   PLI_EC[144] := FALSE;
   PLI_EC[145] := FALSE;
   PLI_EC[146] := FALSE;
   PLI_EC[147] := FALSE;
   PLI_EC[148] := FALSE;
   PLI_EC[149] := FALSE;
   PLI_EC[150] := FALSE;
   PLI_R[1] := FALSE;
   PLI_R[2] := FALSE;
   PLI_R[3] := FALSE;
   PLI_R[4] := FALSE;
   PLI_R[5] := FALSE;
   PLI_R[6] := FALSE;
   PLI_R[7] := FALSE;
   PLI_R[8] := FALSE;
   PLI_R[9] := FALSE;
   PLI_R[10] := FALSE;
   PLI_R[11] := FALSE;
   PLI_R[12] := FALSE;
   PLI_R[13] := FALSE;
   PLI_R[14] := FALSE;
   PLI_R[15] := FALSE;
   PLI_R[16] := FALSE;
   PLI_R[17] := FALSE;
   PLI_R[18] := FALSE;
   PLI_R[19] := FALSE;
   PLI_R[20] := FALSE;
   PLI_R[21] := FALSE;
   PLI_R[22] := FALSE;
   PLI_R[23] := FALSE;
   PLI_R[24] := FALSE;
   PLI_R[25] := FALSE;
   PLI_R[26] := FALSE;
   PLI_R[27] := FALSE;
   PLI_R[28] := FALSE;
   PLI_R[29] := FALSE;
   PLI_R[30] := FALSE;
   PLI_R[31] := FALSE;
   PLI_R[32] := FALSE;
   PLI_R[33] := FALSE;
   PLI_R[34] := FALSE;
   PLI_R[35] := FALSE;
   PLI_R[36] := FALSE;
   PLI_R[37] := FALSE;
   PLI_R[38] := FALSE;
   PLI_R[39] := FALSE;
   PLI_R[40] := FALSE;
   PLI_R[41] := FALSE;
   PLI_R[42] := FALSE;
   PLI_R[43] := FALSE;
   PLI_R[44] := TRUE;
   PLI_R[45] := FALSE;
   PLI_R[46] := FALSE;
   PLI_R[47] := FALSE;
   PLI_R[48] := FALSE;
   PLI_R[49] := FALSE;
   PLI_R[50] := FALSE;
   PLI_R[51] := FALSE;
   PLI_R[52] := FALSE;
   PLI_R[53] := FALSE;
   PLI_R[54] := FALSE;
   PLI_R[55] := FALSE;
   PLI_R[56] := FALSE;
   PLI_R[57] := FALSE;
   PLI_R[58] := FALSE;
   PLI_R[59] := FALSE;
   PLI_R[60] := FALSE;
   PLI_R[61] := FALSE;
   PLI_R[62] := FALSE;
   PLI_R[63] := FALSE;
   PLI_R[64] := FALSE;
   PLI_R[65] := FALSE;
   PLI_R[66] := FALSE;
   PLI_R[67] := FALSE;
   PLI_R[68] := FALSE;
   PLI_R[69] := FALSE;
   PLI_R[70] := FALSE;
   PLI_R[71] := FALSE;
   PLI_R[72] := FALSE;
   PLI_R[73] := FALSE;
   PLI_R[74] := FALSE;
   PLI_R[75] := FALSE;
   PLI_R[76] := FALSE;
   PLI_R[77] := FALSE;
   PLI_R[78] := FALSE;
   PLI_R[79] := FALSE;
   PLI_R[80] := FALSE;
   PLI_R[81] := FALSE;
   PLI_R[82] := FALSE;
   PLI_R[83] := FALSE;
   PLI_R[84] := FALSE;
   PLI_R[85] := FALSE;
   PLI_R[86] := FALSE;
   PLI_R[87] := FALSE;
   PLI_R[88] := FALSE;
   PLI_R[89] := FALSE;
   PLI_R[90] := FALSE;
   PLI_R[91] := FALSE;
   PLI_R[92] := FALSE;
   PLI_R[93] := FALSE;
   PLI_R[94] := FALSE;
   PLI_R[95] := FALSE;
   PLI_R[96] := FALSE;
   PLI_R[97] := FALSE;
   PLI_R[98] := FALSE;
   PLI_R[99] := FALSE;
   PLI_R[100] := FALSE;
   PLI_R[101] := FALSE;
   PLI_R[102] := FALSE;
   PLI_R[103] := FALSE;
   PLI_R[104] := FALSE;
   PLI_R[105] := FALSE;
   PLI_R[106] := FALSE;
   PLI_R[107] := FALSE;
   PLI_R[108] := FALSE;
   PLI_R[109] := FALSE;
   PLI_R[110] := TRUE;
   PLI_R[111] := TRUE;
   PLI_R[112] := FALSE;
   PLI_R[113] := FALSE;
   PLI_R[114] := FALSE;
   PLI_R[115] := FALSE;
   PLI_R[116] := TRUE;
   PLI_R[117] := FALSE;
   PLI_R[118] := FALSE;
   PLI_R[119] := FALSE;
   PLI_R[120] := FALSE;
   PLI_R[121] := FALSE;
   PLI_R[122] := FALSE;
   PLI_R[123] := FALSE;
   PLI_R[124] := FALSE;
   PLI_R[125] := FALSE;
   PLI_R[126] := FALSE;
   PLI_R[127] := FALSE;
   PLI_R[128] := FALSE;
   PLI_R[129] := FALSE;
   PLI_R[130] := FALSE;
   PLI_R[131] := FALSE;
   PLI_R[132] := FALSE;
   PLI_R[133] := FALSE;
   PLI_R[134] := FALSE;
   PLI_R[135] := FALSE;
   PLI_R[136] := FALSE;
   PLI_R[137] := FALSE;
   PLI_R[138] := FALSE;
   PLI_R[139] := FALSE;
   PLI_R[140] := FALSE;
   PLI_R[141] := FALSE;
   PLI_R[142] := FALSE;
   PLI_R[143] := FALSE;
   PLI_R[144] := FALSE;
   PLI_R[145] := FALSE;
   PLI_R[146] := FALSE;
   PLI_R[147] := FALSE;
   PLI_R[148] := FALSE;
   PLI_R[149] := FALSE;
   PLI_R[150] := FALSE;
   PLI_T[1] := FALSE;
   PLI_T[2] := FALSE;
   PLI_T[3] := FALSE;
   PLI_T[4] := FALSE;
   PLI_T[5] := FALSE;
   PLI_T[6] := FALSE;
   PLI_T[7] := FALSE;
   PLI_T[8] := FALSE;
   PLI_T[9] := FALSE;
   PLI_T[10] := FALSE;
   PLI_T[11] := FALSE;
   PLI_T[12] := FALSE;
   PLI_T[13] := FALSE;
   PLI_T[14] := FALSE;
   PLI_T[15] := FALSE;
   PLI_T[16] := FALSE;
   PLI_T[17] := FALSE;
   PLI_T[18] := FALSE;
   PLI_T[19] := FALSE;
   PLI_T[20] := FALSE;
   PLI_T[21] := FALSE;
   PLI_T[22] := FALSE;
   PLI_T[23] := FALSE;
   PLI_T[24] := FALSE;
   PLI_T[25] := FALSE;
   PLI_T[26] := FALSE;
   PLI_T[27] := FALSE;
   PLI_T[28] := FALSE;
   PLI_T[29] := FALSE;
   PLI_T[30] := FALSE;
   PLI_T[31] := FALSE;
   PLI_T[32] := FALSE;
   PLI_T[33] := FALSE;
   PLI_T[34] := FALSE;
   PLI_T[35] := FALSE;
   PLI_T[36] := FALSE;
   PLI_T[37] := FALSE;
   PLI_T[38] := FALSE;
   PLI_T[39] := FALSE;
   PLI_T[40] := FALSE;
   PLI_T[41] := FALSE;
   PLI_T[42] := FALSE;
   PLI_T[43] := FALSE;
   PLI_T[44] := FALSE;
   PLI_T[45] := FALSE;
   PLI_T[46] := FALSE;
   PLI_T[47] := FALSE;
   PLI_T[48] := FALSE;
   PLI_T[49] := FALSE;
   PLI_T[50] := FALSE;
   PLI_T[51] := FALSE;
   PLI_T[52] := FALSE;
   PLI_T[53] := FALSE;
   PLI_T[54] := FALSE;
   PLI_T[55] := FALSE;
   PLI_T[56] := FALSE;
   PLI_T[57] := FALSE;
   PLI_T[58] := FALSE;
   PLI_T[59] := FALSE;
   PLI_T[60] := FALSE;
   PLI_T[61] := FALSE;
   PLI_T[62] := FALSE;
   PLI_T[63] := FALSE;
   PLI_T[64] := FALSE;
   PLI_T[65] := FALSE;
   PLI_T[66] := FALSE;
   PLI_T[67] := FALSE;
   PLI_T[68] := FALSE;
   PLI_T[69] := FALSE;
   PLI_T[70] := FALSE;
   PLI_T[71] := FALSE;
   PLI_T[72] := FALSE;
   PLI_T[73] := FALSE;
   PLI_T[74] := FALSE;
   PLI_T[75] := FALSE;
   PLI_T[76] := FALSE;
   PLI_T[77] := FALSE;
   PLI_T[78] := FALSE;
   PLI_T[79] := FALSE;
   PLI_T[80] := FALSE;
   PLI_T[81] := FALSE;
   PLI_T[82] := FALSE;
   PLI_T[83] := FALSE;
   PLI_T[84] := FALSE;
   PLI_T[85] := FALSE;
   PLI_T[86] := FALSE;
   PLI_T[87] := FALSE;
   PLI_T[88] := FALSE;
   PLI_T[89] := FALSE;
   PLI_T[90] := FALSE;
   PLI_T[91] := FALSE;
   PLI_T[92] := FALSE;
   PLI_T[93] := FALSE;
   PLI_T[94] := FALSE;
   PLI_T[95] := FALSE;
   PLI_T[96] := FALSE;
   PLI_T[97] := FALSE;
   PLI_T[98] := FALSE;
   PLI_T[99] := FALSE;
   PLI_T[100] := FALSE;
   PLI_T[101] := FALSE;
   PLI_T[102] := FALSE;
   PLI_T[103] := FALSE;
   PLI_T[104] := FALSE;
   PLI_T[105] := FALSE;
   PLI_T[106] := FALSE;
   PLI_T[107] := FALSE;
   PLI_T[108] := FALSE;
   PLI_T[109] := FALSE;
   PLI_T[110] := FALSE;
   PLI_T[111] := FALSE;
   PLI_T[112] := FALSE;
   PLI_T[113] := FALSE;
   PLI_T[114] := FALSE;
   PLI_T[115] := FALSE;
   PLI_T[116] := FALSE;
   PLI_T[117] := FALSE;
   PLI_T[118] := FALSE;
   PLI_T[119] := FALSE;
   PLI_T[120] := FALSE;
   PLI_T[121] := FALSE;
   PLI_T[122] := FALSE;
   PLI_T[123] := FALSE;
   PLI_T[124] := FALSE;
   PLI_T[125] := FALSE;
   PLI_T[126] := FALSE;
   PLI_T[127] := FALSE;
   PLI_T[128] := FALSE;
   PLI_T[129] := FALSE;
   PLI_T[130] := FALSE;
   PLI_T[131] := FALSE;
   PLI_T[132] := FALSE;
   PLI_T[133] := FALSE;
   PLI_T[134] := FALSE;
   PLI_T[135] := FALSE;
   PLI_T[136] := FALSE;
   PLI_T[137] := FALSE;
   PLI_T[138] := FALSE;
   PLI_T[139] := FALSE;
   PLI_T[140] := FALSE;
   PLI_T[141] := FALSE;
   PLI_T[142] := FALSE;
   PLI_T[143] := FALSE;
   PLI_T[144] := FALSE;
   PLI_T[145] := FALSE;
   PLI_T[146] := FALSE;
   PLI_T[147] := FALSE;
   PLI_T[148] := FALSE;
   PLI_T[149] := FALSE;
   PLI_T[150] := FALSE;
   PLI_A[1] := FALSE;
   PLI_A[2] := FALSE;
   PLI_A[3] := FALSE;
   PLI_A[4] := FALSE;
   PLI_A[5] := FALSE;
   PLI_A[6] := FALSE;
   PLI_A[7] := FALSE;
   PLI_A[8] := FALSE;
   PLI_A[9] := FALSE;
   PLI_A[10] := FALSE;
   PLI_A[11] := FALSE;
   PLI_A[12] := FALSE;
   PLI_A[13] := FALSE;
   PLI_A[14] := FALSE;
   PLI_A[15] := FALSE;
   PLI_A[16] := FALSE;
   PLI_A[17] := FALSE;
   PLI_A[18] := FALSE;
   PLI_A[19] := FALSE;
   PLI_A[20] := FALSE;
   PLI_A[21] := FALSE;
   PLI_A[22] := FALSE;
   PLI_A[23] := FALSE;
   PLI_A[24] := FALSE;
   PLI_A[25] := FALSE;
   PLI_A[26] := FALSE;
   PLI_A[27] := FALSE;
   PLI_A[28] := FALSE;
   PLI_A[29] := FALSE;
   PLI_A[30] := FALSE;
   PLI_A[31] := FALSE;
   PLI_A[32] := FALSE;
   PLI_A[33] := FALSE;
   PLI_A[34] := FALSE;
   PLI_A[35] := FALSE;
   PLI_A[36] := FALSE;
   PLI_A[37] := FALSE;
   PLI_A[38] := FALSE;
   PLI_A[39] := FALSE;
   PLI_A[40] := FALSE;
   PLI_A[41] := FALSE;
   PLI_A[42] := FALSE;
   PLI_A[43] := FALSE;
   PLI_A[44] := FALSE;
   PLI_A[45] := FALSE;
   PLI_A[46] := FALSE;
   PLI_A[47] := FALSE;
   PLI_A[48] := FALSE;
   PLI_A[49] := FALSE;
   PLI_A[50] := FALSE;
   PLI_A[51] := FALSE;
   PLI_A[52] := FALSE;
   PLI_A[53] := FALSE;
   PLI_A[54] := FALSE;
   PLI_A[55] := FALSE;
   PLI_A[56] := FALSE;
   PLI_A[57] := FALSE;
   PLI_A[58] := FALSE;
   PLI_A[59] := FALSE;
   PLI_A[60] := FALSE;
   PLI_A[61] := FALSE;
   PLI_A[62] := FALSE;
   PLI_A[63] := FALSE;
   PLI_A[64] := FALSE;
   PLI_A[65] := FALSE;
   PLI_A[66] := FALSE;
   PLI_A[67] := FALSE;
   PLI_A[68] := FALSE;
   PLI_A[69] := FALSE;
   PLI_A[70] := FALSE;
   PLI_A[71] := FALSE;
   PLI_A[72] := FALSE;
   PLI_A[73] := FALSE;
   PLI_A[74] := FALSE;
   PLI_A[75] := FALSE;
   PLI_A[76] := FALSE;
   PLI_A[77] := FALSE;
   PLI_A[78] := FALSE;
   PLI_A[79] := FALSE;
   PLI_A[80] := FALSE;
   PLI_A[81] := FALSE;
   PLI_A[82] := FALSE;
   PLI_A[83] := FALSE;
   PLI_A[84] := FALSE;
   PLI_A[85] := FALSE;
   PLI_A[86] := FALSE;
   PLI_A[87] := FALSE;
   PLI_A[88] := FALSE;
   PLI_A[89] := FALSE;
   PLI_A[90] := FALSE;
   PLI_A[91] := FALSE;
   PLI_A[92] := FALSE;
   PLI_A[93] := FALSE;
   PLI_A[94] := FALSE;
   PLI_A[95] := FALSE;
   PLI_A[96] := FALSE;
   PLI_A[97] := FALSE;
   PLI_A[98] := FALSE;
   PLI_A[99] := FALSE;
   PLI_A[100] := FALSE;
   PLI_A[101] := FALSE;
   PLI_A[102] := FALSE;
   PLI_A[103] := FALSE;
   PLI_A[104] := FALSE;
   PLI_A[105] := FALSE;
   PLI_A[106] := FALSE;
   PLI_A[107] := FALSE;
   PLI_A[108] := FALSE;
   PLI_A[109] := FALSE;
   PLI_A[110] := FALSE;
   PLI_A[111] := FALSE;
   PLI_A[112] := FALSE;
   PLI_A[113] := FALSE;
   PLI_A[114] := FALSE;
   PLI_A[115] := FALSE;
   PLI_A[116] := FALSE;
   PLI_A[117] := FALSE;
   PLI_A[118] := FALSE;
   PLI_A[119] := FALSE;
   PLI_A[120] := FALSE;
   PLI_A[121] := FALSE;
   PLI_A[122] := FALSE;
   PLI_A[123] := FALSE;
   PLI_A[124] := FALSE;
   PLI_A[125] := FALSE;
   PLI_A[126] := FALSE;
   PLI_A[127] := FALSE;
   PLI_A[128] := FALSE;
   PLI_A[129] := FALSE;
   PLI_A[130] := FALSE;
   PLI_A[131] := FALSE;
   PLI_A[132] := FALSE;
   PLI_A[133] := FALSE;
   PLI_A[134] := FALSE;
   PLI_A[135] := FALSE;
   PLI_A[136] := FALSE;
   PLI_A[137] := FALSE;
   PLI_A[138] := FALSE;
   PLI_A[139] := FALSE;
   PLI_A[140] := FALSE;
   PLI_A[141] := FALSE;
   PLI_A[142] := FALSE;
   PLI_A[143] := FALSE;
   PLI_A[144] := FALSE;
   PLI_A[145] := FALSE;
   PLI_A[146] := FALSE;
   PLI_A[147] := FALSE;
   PLI_A[148] := FALSE;
   PLI_A[149] := FALSE;
   PLI_A[150] := FALSE;
   PLI_H[1] := FALSE;
   PLI_H[2] := FALSE;
   PLI_H[3] := FALSE;
   PLI_H[4] := FALSE;
   PLI_H[5] := FALSE;
   PLI_H[6] := FALSE;
   PLI_H[7] := FALSE;
   PLI_H[8] := FALSE;
   PLI_H[9] := FALSE;
   PLI_H[10] := FALSE;
   PLI_H[11] := FALSE;
   PLI_H[12] := FALSE;
   PLI_H[13] := FALSE;
   PLI_H[14] := FALSE;
   PLI_H[15] := FALSE;
   PLI_H[16] := FALSE;
   PLI_H[17] := FALSE;
   PLI_H[18] := FALSE;
   PLI_H[19] := FALSE;
   PLI_H[20] := FALSE;
   PLI_H[21] := FALSE;
   PLI_H[22] := FALSE;
   PLI_H[23] := FALSE;
   PLI_H[24] := FALSE;
   PLI_H[25] := FALSE;
   PLI_H[26] := FALSE;
   PLI_H[27] := FALSE;
   PLI_H[28] := FALSE;
   PLI_H[29] := FALSE;
   PLI_H[30] := FALSE;
   PLI_H[31] := FALSE;
   PLI_H[32] := FALSE;
   PLI_H[33] := FALSE;
   PLI_H[34] := FALSE;
   PLI_H[35] := FALSE;
   PLI_H[36] := FALSE;
   PLI_H[37] := FALSE;
   PLI_H[38] := FALSE;
   PLI_H[39] := FALSE;
   PLI_H[40] := FALSE;
   PLI_H[41] := FALSE;
   PLI_H[42] := FALSE;
   PLI_H[43] := FALSE;
   PLI_H[44] := FALSE;
   PLI_H[45] := FALSE;
   PLI_H[46] := FALSE;
   PLI_H[47] := FALSE;
   PLI_H[48] := FALSE;
   PLI_H[49] := FALSE;
   PLI_H[50] := FALSE;
   PLI_H[51] := FALSE;
   PLI_H[52] := FALSE;
   PLI_H[53] := FALSE;
   PLI_H[54] := FALSE;
   PLI_H[55] := FALSE;
   PLI_H[56] := FALSE;
   PLI_H[57] := FALSE;
   PLI_H[58] := FALSE;
   PLI_H[59] := FALSE;
   PLI_H[60] := FALSE;
   PLI_H[61] := FALSE;
   PLI_H[62] := FALSE;
   PLI_H[63] := FALSE;
   PLI_H[64] := FALSE;
   PLI_H[65] := FALSE;
   PLI_H[66] := FALSE;
   PLI_H[67] := FALSE;
   PLI_H[68] := FALSE;
   PLI_H[69] := FALSE;
   PLI_H[70] := FALSE;
   PLI_H[71] := FALSE;
   PLI_H[72] := FALSE;
   PLI_H[73] := FALSE;
   PLI_H[74] := FALSE;
   PLI_H[75] := FALSE;
   PLI_H[76] := FALSE;
   PLI_H[77] := FALSE;
   PLI_H[78] := FALSE;
   PLI_H[79] := FALSE;
   PLI_H[80] := FALSE;
   PLI_H[81] := FALSE;
   PLI_H[82] := FALSE;
   PLI_H[83] := FALSE;
   PLI_H[84] := FALSE;
   PLI_H[85] := FALSE;
   PLI_H[86] := FALSE;
   PLI_H[87] := FALSE;
   PLI_H[88] := FALSE;
   PLI_H[89] := FALSE;
   PLI_H[90] := FALSE;
   PLI_H[91] := FALSE;
   PLI_H[92] := FALSE;
   PLI_H[93] := FALSE;
   PLI_H[94] := FALSE;
   PLI_H[95] := FALSE;
   PLI_H[96] := FALSE;
   PLI_H[97] := FALSE;
   PLI_H[98] := TRUE;
   PLI_H[99] := FALSE;
   PLI_H[100] := FALSE;
   PLI_H[101] := FALSE;
   PLI_H[102] := FALSE;
   PLI_H[103] := FALSE;
   PLI_H[104] := FALSE;
   PLI_H[105] := FALSE;
   PLI_H[106] := FALSE;
   PLI_H[107] := FALSE;
   PLI_H[108] := FALSE;
   PLI_H[109] := FALSE;
   PLI_H[110] := FALSE;
   PLI_H[111] := FALSE;
   PLI_H[112] := TRUE;
   PLI_H[113] := FALSE;
   PLI_H[114] := FALSE;
   PLI_H[115] := TRUE;
   PLI_H[116] := FALSE;
   PLI_H[117] := FALSE;
   PLI_H[118] := FALSE;
   PLI_H[119] := FALSE;
   PLI_H[120] := FALSE;
   PLI_H[121] := FALSE;
   PLI_H[122] := FALSE;
   PLI_H[123] := FALSE;
   PLI_H[124] := FALSE;
   PLI_H[125] := FALSE;
   PLI_H[126] := FALSE;
   PLI_H[127] := FALSE;
   PLI_H[128] := FALSE;
   PLI_H[129] := FALSE;
   PLI_H[130] := FALSE;
   PLI_H[131] := FALSE;
   PLI_H[132] := FALSE;
   PLI_H[133] := FALSE;
   PLI_H[134] := FALSE;
   PLI_H[135] := FALSE;
   PLI_H[136] := FALSE;
   PLI_H[137] := FALSE;
   PLI_H[138] := FALSE;
   PLI_H[139] := FALSE;
   PLI_H[140] := FALSE;
   PLI_H[141] := FALSE;
   PLI_H[142] := FALSE;
   PLI_H[143] := FALSE;
   PLI_H[144] := FALSE;
   PLI_H[145] := FALSE;
   PLI_H[146] := FALSE;
   PLI_H[147] := FALSE;
   PLI_H[148] := FALSE;
   PLI_H[149] := FALSE;
   PLI_H[150] := FALSE;
   PLI_S[1] := FALSE;
   PLI_S[2] := FALSE;
   PLI_S[3] := FALSE;
   PLI_S[4] := FALSE;
   PLI_S[5] := FALSE;
   PLI_S[6] := FALSE;
   PLI_S[7] := FALSE;
   PLI_S[8] := FALSE;
   PLI_S[9] := FALSE;
   PLI_S[10] := FALSE;
   PLI_S[11] := FALSE;
   PLI_S[12] := FALSE;
   PLI_S[13] := FALSE;
   PLI_S[14] := FALSE;
   PLI_S[15] := FALSE;
   PLI_S[16] := FALSE;
   PLI_S[17] := FALSE;
   PLI_S[18] := FALSE;
   PLI_S[19] := FALSE;
   PLI_S[20] := FALSE;
   PLI_S[21] := FALSE;
   PLI_S[22] := FALSE;
   PLI_S[23] := FALSE;
   PLI_S[24] := FALSE;
   PLI_S[25] := FALSE;
   PLI_S[26] := FALSE;
   PLI_S[27] := FALSE;
   PLI_S[28] := FALSE;
   PLI_S[29] := FALSE;
   PLI_S[30] := FALSE;
   PLI_S[31] := FALSE;
   PLI_S[32] := FALSE;
   PLI_S[33] := FALSE;
   PLI_S[34] := FALSE;
   PLI_S[35] := FALSE;
   PLI_S[36] := FALSE;
   PLI_S[37] := FALSE;
   PLI_S[38] := FALSE;
   PLI_S[39] := FALSE;
   PLI_S[40] := FALSE;
   PLI_S[41] := FALSE;
   PLI_S[42] := FALSE;
   PLI_S[43] := FALSE;
   PLI_S[44] := FALSE;
   PLI_S[45] := FALSE;
   PLI_S[46] := FALSE;
   PLI_S[47] := FALSE;
   PLI_S[48] := FALSE;
   PLI_S[49] := FALSE;
   PLI_S[50] := FALSE;
   PLI_S[51] := FALSE;
   PLI_S[52] := FALSE;
   PLI_S[53] := FALSE;
   PLI_S[54] := FALSE;
   PLI_S[55] := FALSE;
   PLI_S[56] := FALSE;
   PLI_S[57] := FALSE;
   PLI_S[58] := FALSE;
   PLI_S[59] := FALSE;
   PLI_S[60] := FALSE;
   PLI_S[61] := FALSE;
   PLI_S[62] := FALSE;
   PLI_S[63] := FALSE;
   PLI_S[64] := FALSE;
   PLI_S[65] := FALSE;
   PLI_S[66] := FALSE;
   PLI_S[67] := FALSE;
   PLI_S[68] := FALSE;
   PLI_S[69] := FALSE;
   PLI_S[70] := FALSE;
   PLI_S[71] := FALSE;
   PLI_S[72] := FALSE;
   PLI_S[73] := FALSE;
   PLI_S[74] := FALSE;
   PLI_S[75] := FALSE;
   PLI_S[76] := FALSE;
   PLI_S[77] := FALSE;
   PLI_S[78] := FALSE;
   PLI_S[79] := FALSE;
   PLI_S[80] := FALSE;
   PLI_S[81] := FALSE;
   PLI_S[82] := FALSE;
   PLI_S[83] := FALSE;
   PLI_S[84] := FALSE;
   PLI_S[85] := FALSE;
   PLI_S[86] := FALSE;
   PLI_S[87] := FALSE;
   PLI_S[88] := FALSE;
   PLI_S[89] := FALSE;
   PLI_S[90] := FALSE;
   PLI_S[91] := FALSE;
   PLI_S[92] := FALSE;
   PLI_S[93] := FALSE;
   PLI_S[94] := FALSE;
   PLI_S[95] := FALSE;
   PLI_S[96] := FALSE;
   PLI_S[97] := FALSE;
   PLI_S[98] := FALSE;
   PLI_S[99] := FALSE;
   PLI_S[100] := FALSE;
   PLI_S[101] := FALSE;
   PLI_S[102] := FALSE;
   PLI_S[103] := FALSE;
   PLI_S[104] := FALSE;
   PLI_S[105] := FALSE;
   PLI_S[106] := FALSE;
   PLI_S[107] := FALSE;
   PLI_S[108] := FALSE;
   PLI_S[109] := FALSE;
   PLI_S[110] := FALSE;
   PLI_S[111] := FALSE;
   PLI_S[112] := FALSE;
   PLI_S[113] := FALSE;
   PLI_S[114] := FALSE;
   PLI_S[115] := FALSE;
   PLI_S[116] := FALSE;
   PLI_S[117] := FALSE;
   PLI_S[118] := FALSE;
   PLI_S[119] := FALSE;
   PLI_S[120] := FALSE;
   PLI_S[121] := FALSE;
   PLI_S[122] := FALSE;
   PLI_S[123] := FALSE;
   PLI_S[124] := FALSE;
   PLI_S[125] := FALSE;
   PLI_S[126] := FALSE;
   PLI_S[127] := FALSE;
   PLI_S[128] := FALSE;
   PLI_S[129] := FALSE;
   PLI_S[130] := FALSE;
   PLI_S[131] := FALSE;
   PLI_S[132] := FALSE;
   PLI_S[133] := FALSE;
   PLI_S[134] := FALSE;
   PLI_S[135] := FALSE;
   PLI_S[136] := FALSE;
   PLI_S[137] := FALSE;
   PLI_S[138] := FALSE;
   PLI_S[139] := FALSE;
   PLI_S[140] := FALSE;
   PLI_S[141] := FALSE;
   PLI_S[142] := FALSE;
   PLI_S[143] := FALSE;
   PLI_S[144] := FALSE;
   PLI_S[145] := FALSE;
   PLI_S[146] := FALSE;
   PLI_S[147] := FALSE;
   PLI_S[148] := FALSE;
   PLI_S[149] := FALSE;
   PLI_S[150] := FALSE;
   PLI_E[1] := TRUE;
   PLI_E[2] := TRUE;
   PLI_E[3] := TRUE;
   PLI_E[4] := TRUE;
   PLI_E[5] := TRUE;
   PLI_E[6] := TRUE;
   PLI_E[7] := TRUE;
   PLI_E[8] := TRUE;
   PLI_E[9] := TRUE;
   PLI_E[10] := TRUE;
   PLI_E[11] := TRUE;
   PLI_E[12] := TRUE;
   PLI_E[13] := TRUE;
   PLI_E[14] := TRUE;
   PLI_E[15] := TRUE;
   PLI_E[16] := TRUE;
   PLI_E[17] := TRUE;
   PLI_E[18] := TRUE;
   PLI_E[19] := TRUE;
   PLI_E[20] := TRUE;
   PLI_E[21] := TRUE;
   PLI_E[22] := TRUE;
   PLI_E[23] := TRUE;
   PLI_E[24] := TRUE;
   PLI_E[25] := TRUE;
   PLI_E[26] := TRUE;
   PLI_E[27] := TRUE;
   PLI_E[28] := TRUE;
   PLI_E[29] := TRUE;
   PLI_E[30] := TRUE;
   PLI_E[31] := TRUE;
   PLI_E[32] := TRUE;
   PLI_E[33] := TRUE;
   PLI_E[34] := TRUE;
   PLI_E[35] := TRUE;
   PLI_E[36] := TRUE;
   PLI_E[37] := TRUE;
   PLI_E[38] := TRUE;
   PLI_E[39] := TRUE;
   PLI_E[40] := TRUE;
   PLI_E[41] := TRUE;
   PLI_E[42] := TRUE;
   PLI_E[43] := TRUE;
   PLI_E[44] := FALSE;
   PLI_E[45] := TRUE;
   PLI_E[46] := TRUE;
   PLI_E[47] := TRUE;
   PLI_E[48] := TRUE;
   PLI_E[49] := TRUE;
   PLI_E[50] := TRUE;
   PLI_E[51] := TRUE;
   PLI_E[52] := TRUE;
   PLI_E[53] := TRUE;
   PLI_E[54] := TRUE;
   PLI_E[55] := TRUE;
   PLI_E[56] := FALSE;
   PLI_E[57] := TRUE;
   PLI_E[58] := TRUE;
   PLI_E[59] := TRUE;
   PLI_E[60] := TRUE;
   PLI_E[61] := TRUE;
   PLI_E[62] := TRUE;
   PLI_E[63] := TRUE;
   PLI_E[64] := TRUE;
   PLI_E[65] := TRUE;
   PLI_E[66] := FALSE;
   PLI_E[67] := FALSE;
   PLI_E[68] := TRUE;
   PLI_E[69] := TRUE;
   PLI_E[70] := TRUE;
   PLI_E[71] := TRUE;
   PLI_E[72] := TRUE;
   PLI_E[73] := FALSE;
   PLI_E[74] := TRUE;
   PLI_E[75] := TRUE;
   PLI_E[76] := FALSE;
   PLI_E[77] := TRUE;
   PLI_E[78] := TRUE;
   PLI_E[79] := TRUE;
   PLI_E[80] := TRUE;
   PLI_E[81] := TRUE;
   PLI_E[82] := TRUE;
   PLI_E[83] := TRUE;
   PLI_E[84] := TRUE;
   PLI_E[85] := TRUE;
   PLI_E[86] := TRUE;
   PLI_E[87] := TRUE;
   PLI_E[88] := TRUE;
   PLI_E[89] := TRUE;
   PLI_E[90] := TRUE;
   PLI_E[91] := TRUE;
   PLI_E[92] := TRUE;
   PLI_E[93] := TRUE;
   PLI_E[94] := TRUE;
   PLI_E[95] := TRUE;
   PLI_E[96] := TRUE;
   PLI_E[97] := FALSE;
   PLI_E[98] := FALSE;
   PLI_E[99] := FALSE;
   PLI_E[100] := TRUE;
   PLI_E[101] := TRUE;
   PLI_E[102] := TRUE;
   PLI_E[103] := TRUE;
   PLI_E[104] := FALSE;
   PLI_E[105] := TRUE;
   PLI_E[106] := FALSE;
   PLI_E[107] := FALSE;
   PLI_E[108] := FALSE;
   PLI_E[109] := FALSE;
   PLI_E[110] := FALSE;
   PLI_E[111] := FALSE;
   PLI_E[112] := FALSE;
   PLI_E[113] := FALSE;
   PLI_E[114] := FALSE;
   PLI_E[115] := FALSE;
   PLI_E[116] := FALSE;
   PLI_E[117] := FALSE;
   PLI_E[118] := FALSE;
   PLI_E[119] := FALSE;
   PLI_E[120] := TRUE;
   PLI_E[121] := TRUE;
   PLI_E[122] := TRUE;
   PLI_E[123] := FALSE;
   PLI_E[124] := FALSE;
   PLI_E[125] := FALSE;
   PLI_E[126] := FALSE;
   PLI_E[127] := FALSE;
   PLI_E[128] := FALSE;
   PLI_E[129] := FALSE;
   PLI_E[130] := FALSE;
   PLI_E[131] := FALSE;
   PLI_E[132] := FALSE;
   PLI_E[133] := FALSE;
   PLI_E[134] := FALSE;
   PLI_E[135] := FALSE;
   PLI_E[136] := FALSE;
   PLI_E[137] := FALSE;
   PLI_E[138] := FALSE;
   PLI_E[139] := FALSE;
   PLI_E[140] := FALSE;
   PLI_E[141] := FALSE;
   PLI_E[142] := FALSE;
   PLI_E[143] := FALSE;
   PLI_E[144] := FALSE;
   PLI_E[145] := FALSE;
   PLI_E[146] := FALSE;
   PLI_E[147] := FALSE;
   PLI_E[148] := FALSE;
   PLI_E[149] := FALSE;
   PLI_E[150] := FALSE;
   PLI_I[1] := TRUE;
   PLI_I[2] := TRUE;
   PLI_I[3] := TRUE;
   PLI_I[4] := TRUE;
   PLI_I[5] := TRUE;
   PLI_I[6] := TRUE;
   PLI_I[7] := TRUE;
   PLI_I[8] := TRUE;
   PLI_I[9] := TRUE;
   PLI_I[10] := TRUE;
   PLI_I[11] := TRUE;
   PLI_I[12] := TRUE;
   PLI_I[13] := TRUE;
   PLI_I[14] := TRUE;
   PLI_I[15] := TRUE;
   PLI_I[16] := TRUE;
   PLI_I[17] := TRUE;
   PLI_I[18] := TRUE;
   PLI_I[19] := TRUE;
   PLI_I[20] := TRUE;
   PLI_I[21] := TRUE;
   PLI_I[22] := TRUE;
   PLI_I[23] := TRUE;
   PLI_I[24] := TRUE;
   PLI_I[25] := TRUE;
   PLI_I[26] := TRUE;
   PLI_I[27] := TRUE;
   PLI_I[28] := TRUE;
   PLI_I[29] := TRUE;
   PLI_I[30] := TRUE;
   PLI_I[31] := TRUE;
   PLI_I[32] := TRUE;
   PLI_I[33] := TRUE;
   PLI_I[34] := TRUE;
   PLI_I[35] := TRUE;
   PLI_I[36] := TRUE;
   PLI_I[37] := TRUE;
   PLI_I[38] := TRUE;
   PLI_I[39] := TRUE;
   PLI_I[40] := TRUE;
   PLI_I[41] := TRUE;
   PLI_I[42] := TRUE;
   PLI_I[43] := TRUE;
   PLI_I[44] := TRUE;
   PLI_I[45] := TRUE;
   PLI_I[46] := TRUE;
   PLI_I[47] := TRUE;
   PLI_I[48] := TRUE;
   PLI_I[49] := TRUE;
   PLI_I[50] := TRUE;
   PLI_I[51] := TRUE;
   PLI_I[52] := TRUE;
   PLI_I[53] := TRUE;
   PLI_I[54] := TRUE;
   PLI_I[55] := TRUE;
   PLI_I[56] := TRUE;
   PLI_I[57] := TRUE;
   PLI_I[58] := TRUE;
   PLI_I[59] := TRUE;
   PLI_I[60] := TRUE;
   PLI_I[61] := TRUE;
   PLI_I[62] := TRUE;
   PLI_I[63] := TRUE;
   PLI_I[64] := TRUE;
   PLI_I[65] := TRUE;
   PLI_I[66] := TRUE;
   PLI_I[67] := TRUE;
   PLI_I[68] := TRUE;
   PLI_I[69] := TRUE;
   PLI_I[70] := TRUE;
   PLI_I[71] := TRUE;
   PLI_I[72] := TRUE;
   PLI_I[73] := TRUE;
   PLI_I[74] := TRUE;
   PLI_I[75] := TRUE;
   PLI_I[76] := TRUE;
   PLI_I[77] := TRUE;
   PLI_I[78] := TRUE;
   PLI_I[79] := TRUE;
   PLI_I[80] := TRUE;
   PLI_I[81] := TRUE;
   PLI_I[82] := TRUE;
   PLI_I[83] := TRUE;
   PLI_I[84] := TRUE;
   PLI_I[85] := TRUE;
   PLI_I[86] := TRUE;
   PLI_I[87] := TRUE;
   PLI_I[88] := TRUE;
   PLI_I[89] := TRUE;
   PLI_I[90] := TRUE;
   PLI_I[91] := TRUE;
   PLI_I[92] := TRUE;
   PLI_I[93] := TRUE;
   PLI_I[94] := TRUE;
   PLI_I[95] := TRUE;
   PLI_I[96] := TRUE;
   PLI_I[97] := TRUE;
   PLI_I[98] := TRUE;
   PLI_I[99] := TRUE;
   PLI_I[100] := TRUE;
   PLI_I[101] := TRUE;
   PLI_I[102] := TRUE;
   PLI_I[103] := TRUE;
   PLI_I[104] := TRUE;
   PLI_I[105] := TRUE;
   PLI_I[106] := TRUE;
   PLI_I[107] := TRUE;
   PLI_I[108] := TRUE;
   PLI_I[109] := TRUE;
   PLI_I[110] := FALSE;
   PLI_I[111] := FALSE;
   PLI_I[112] := TRUE;
   PLI_I[113] := TRUE;
   PLI_I[114] := TRUE;
   PLI_I[115] := FALSE;
   PLI_I[116] := FALSE;
   PLI_I[117] := TRUE;
   PLI_I[118] := TRUE;
   PLI_I[119] := TRUE;
   PLI_I[120] := TRUE;
   PLI_I[121] := TRUE;
   PLI_I[122] := TRUE;
   PLI_I[123] := TRUE;
   PLI_I[124] := TRUE;
   PLI_I[125] := TRUE;
   PLI_I[126] := TRUE;
   PLI_I[127] := TRUE;
   PLI_I[128] := TRUE;
   PLI_I[129] := TRUE;
   PLI_I[130] := TRUE;
   PLI_I[131] := TRUE;
   PLI_I[132] := TRUE;
   PLI_I[133] := TRUE;
   PLI_I[134] := TRUE;
   PLI_I[135] := TRUE;
   PLI_I[136] := TRUE;
   PLI_I[137] := TRUE;
   PLI_I[138] := TRUE;
   PLI_I[139] := TRUE;
   PLI_I[140] := TRUE;
   PLI_I[141] := TRUE;
   PLI_I[142] := TRUE;
   PLI_I[143] := TRUE;
   PLI_I[144] := TRUE;
   PLI_I[145] := TRUE;
   PLI_I[146] := TRUE;
   PLI_I[147] := TRUE;
   PLI_I[148] := TRUE;
   PLI_I[149] := TRUE;
   PLI_I[150] := TRUE;
   PLI_C[1] := FALSE;
   PLI_C[2] := FALSE;
   PLI_C[3] := FALSE;
   PLI_C[4] := FALSE;
   PLI_C[5] := FALSE;
   PLI_C[6] := FALSE;
   PLI_C[7] := FALSE;
   PLI_C[8] := FALSE;
   PLI_C[9] := FALSE;
   PLI_C[10] := FALSE;
   PLI_C[11] := FALSE;
   PLI_C[12] := FALSE;
   PLI_C[13] := FALSE;
   PLI_C[14] := FALSE;
   PLI_C[15] := FALSE;
   PLI_C[16] := FALSE;
   PLI_C[17] := FALSE;
   PLI_C[18] := FALSE;
   PLI_C[19] := FALSE;
   PLI_C[20] := FALSE;
   PLI_C[21] := FALSE;
   PLI_C[22] := FALSE;
   PLI_C[23] := FALSE;
   PLI_C[24] := FALSE;
   PLI_C[25] := FALSE;
   PLI_C[26] := FALSE;
   PLI_C[27] := FALSE;
   PLI_C[28] := FALSE;
   PLI_C[29] := FALSE;
   PLI_C[30] := FALSE;
   PLI_C[31] := FALSE;
   PLI_C[32] := FALSE;
   PLI_C[33] := FALSE;
   PLI_C[34] := FALSE;
   PLI_C[35] := FALSE;
   PLI_C[36] := FALSE;
   PLI_C[37] := FALSE;
   PLI_C[38] := FALSE;
   PLI_C[39] := FALSE;
   PLI_C[40] := FALSE;
   PLI_C[41] := FALSE;
   PLI_C[42] := FALSE;
   PLI_C[43] := FALSE;
   PLI_C[44] := FALSE;
   PLI_C[45] := FALSE;
   PLI_C[46] := FALSE;
   PLI_C[47] := FALSE;
   PLI_C[48] := FALSE;
   PLI_C[49] := FALSE;
   PLI_C[50] := FALSE;
   PLI_C[51] := FALSE;
   PLI_C[52] := FALSE;
   PLI_C[53] := FALSE;
   PLI_C[54] := FALSE;
   PLI_C[55] := FALSE;
   PLI_C[56] := FALSE;
   PLI_C[57] := FALSE;
   PLI_C[58] := FALSE;
   PLI_C[59] := FALSE;
   PLI_C[60] := FALSE;
   PLI_C[61] := FALSE;
   PLI_C[62] := FALSE;
   PLI_C[63] := FALSE;
   PLI_C[64] := FALSE;
   PLI_C[65] := FALSE;
   PLI_C[66] := FALSE;
   PLI_C[67] := FALSE;
   PLI_C[68] := FALSE;
   PLI_C[69] := FALSE;
   PLI_C[70] := FALSE;
   PLI_C[71] := FALSE;
   PLI_C[72] := FALSE;
   PLI_C[73] := FALSE;
   PLI_C[74] := FALSE;
   PLI_C[75] := FALSE;
   PLI_C[76] := FALSE;
   PLI_C[77] := FALSE;
   PLI_C[78] := FALSE;
   PLI_C[79] := FALSE;
   PLI_C[80] := FALSE;
   PLI_C[81] := FALSE;
   PLI_C[82] := FALSE;
   PLI_C[83] := FALSE;
   PLI_C[84] := FALSE;
   PLI_C[85] := FALSE;
   PLI_C[86] := FALSE;
   PLI_C[87] := FALSE;
   PLI_C[88] := FALSE;
   PLI_C[89] := FALSE;
   PLI_C[90] := FALSE;
   PLI_C[91] := FALSE;
   PLI_C[92] := FALSE;
   PLI_C[93] := FALSE;
   PLI_C[94] := FALSE;
   PLI_C[95] := FALSE;
   PLI_C[96] := FALSE;
   PLI_C[97] := FALSE;
   PLI_C[98] := FALSE;
   PLI_C[99] := FALSE;
   PLI_C[100] := FALSE;
   PLI_C[101] := FALSE;
   PLI_C[102] := FALSE;
   PLI_C[103] := FALSE;
   PLI_C[104] := FALSE;
   PLI_C[105] := FALSE;
   PLI_C[106] := FALSE;
   PLI_C[107] := FALSE;
   PLI_C[108] := FALSE;
   PLI_C[109] := FALSE;
   PLI_C[110] := FALSE;
   PLI_C[111] := FALSE;
   PLI_C[112] := FALSE;
   PLI_C[113] := FALSE;
   PLI_C[114] := FALSE;
   PLI_C[115] := FALSE;
   PLI_C[116] := FALSE;
   PLI_C[117] := FALSE;
   PLI_C[118] := FALSE;
   PLI_C[119] := FALSE;
   PLI_C[120] := FALSE;
   PLI_C[121] := FALSE;
   PLI_C[122] := FALSE;
   PLI_C[123] := FALSE;
   PLI_C[124] := FALSE;
   PLI_C[125] := FALSE;
   PLI_C[126] := FALSE;
   PLI_C[127] := FALSE;
   PLI_C[128] := FALSE;
   PLI_C[129] := FALSE;
   PLI_C[130] := FALSE;
   PLI_C[131] := FALSE;
   PLI_C[132] := FALSE;
   PLI_C[133] := FALSE;
   PLI_C[134] := FALSE;
   PLI_C[135] := FALSE;
   PLI_C[136] := FALSE;
   PLI_C[137] := FALSE;
   PLI_C[138] := FALSE;
   PLI_C[139] := FALSE;
   PLI_C[140] := FALSE;
   PLI_C[141] := FALSE;
   PLI_C[142] := FALSE;
   PLI_C[143] := FALSE;
   PLI_C[144] := FALSE;
   PLI_C[145] := FALSE;
   PLI_C[146] := FALSE;
   PLI_C[147] := FALSE;
   PLI_C[148] := FALSE;
   PLI_C[149] := FALSE;
   PLI_C[150] := FALSE;
   PLI_AD[1] := FALSE;
   PLI_AD[2] := FALSE;
   PLI_AD[3] := FALSE;
   PLI_AD[4] := FALSE;
   PLI_AD[5] := FALSE;
   PLI_AD[6] := FALSE;
   PLI_AD[7] := FALSE;
   PLI_AD[8] := FALSE;
   PLI_AD[9] := FALSE;
   PLI_AD[10] := FALSE;
   PLI_AD[11] := FALSE;
   PLI_AD[12] := FALSE;
   PLI_AD[13] := FALSE;
   PLI_AD[14] := FALSE;
   PLI_AD[15] := FALSE;
   PLI_AD[16] := FALSE;
   PLI_AD[17] := FALSE;
   PLI_AD[18] := FALSE;
   PLI_AD[19] := FALSE;
   PLI_AD[20] := FALSE;
   PLI_AD[21] := FALSE;
   PLI_AD[22] := FALSE;
   PLI_AD[23] := FALSE;
   PLI_AD[24] := FALSE;
   PLI_AD[25] := FALSE;
   PLI_AD[26] := FALSE;
   PLI_AD[27] := FALSE;
   PLI_AD[28] := FALSE;
   PLI_AD[29] := FALSE;
   PLI_AD[30] := FALSE;
   PLI_AD[31] := FALSE;
   PLI_AD[32] := FALSE;
   PLI_AD[33] := FALSE;
   PLI_AD[34] := FALSE;
   PLI_AD[35] := FALSE;
   PLI_AD[36] := FALSE;
   PLI_AD[37] := FALSE;
   PLI_AD[38] := FALSE;
   PLI_AD[39] := FALSE;
   PLI_AD[40] := FALSE;
   PLI_AD[41] := FALSE;
   PLI_AD[42] := FALSE;
   PLI_AD[43] := FALSE;
   PLI_AD[44] := FALSE;
   PLI_AD[45] := FALSE;
   PLI_AD[46] := FALSE;
   PLI_AD[47] := FALSE;
   PLI_AD[48] := FALSE;
   PLI_AD[49] := FALSE;
   PLI_AD[50] := FALSE;
   PLI_AD[51] := FALSE;
   PLI_AD[52] := FALSE;
   PLI_AD[53] := FALSE;
   PLI_AD[54] := FALSE;
   PLI_AD[55] := FALSE;
   PLI_AD[56] := FALSE;
   PLI_AD[57] := FALSE;
   PLI_AD[58] := FALSE;
   PLI_AD[59] := FALSE;
   PLI_AD[60] := FALSE;
   PLI_AD[61] := FALSE;
   PLI_AD[62] := FALSE;
   PLI_AD[63] := FALSE;
   PLI_AD[64] := FALSE;
   PLI_AD[65] := FALSE;
   PLI_AD[66] := FALSE;
   PLI_AD[67] := FALSE;
   PLI_AD[68] := FALSE;
   PLI_AD[69] := FALSE;
   PLI_AD[70] := FALSE;
   PLI_AD[71] := FALSE;
   PLI_AD[72] := FALSE;
   PLI_AD[73] := FALSE;
   PLI_AD[74] := FALSE;
   PLI_AD[75] := FALSE;
   PLI_AD[76] := FALSE;
   PLI_AD[77] := FALSE;
   PLI_AD[78] := FALSE;
   PLI_AD[79] := FALSE;
   PLI_AD[80] := FALSE;
   PLI_AD[81] := FALSE;
   PLI_AD[82] := FALSE;
   PLI_AD[83] := FALSE;
   PLI_AD[84] := FALSE;
   PLI_AD[85] := FALSE;
   PLI_AD[86] := FALSE;
   PLI_AD[87] := FALSE;
   PLI_AD[88] := FALSE;
   PLI_AD[89] := FALSE;
   PLI_AD[90] := FALSE;
   PLI_AD[91] := FALSE;
   PLI_AD[92] := FALSE;
   PLI_AD[93] := FALSE;
   PLI_AD[94] := FALSE;
   PLI_AD[95] := FALSE;
   PLI_AD[96] := FALSE;
   PLI_AD[97] := FALSE;
   PLI_AD[98] := FALSE;
   PLI_AD[99] := FALSE;
   PLI_AD[100] := FALSE;
   PLI_AD[101] := FALSE;
   PLI_AD[102] := FALSE;
   PLI_AD[103] := FALSE;
   PLI_AD[104] := FALSE;
   PLI_AD[105] := FALSE;
   PLI_AD[106] := FALSE;
   PLI_AD[107] := FALSE;
   PLI_AD[108] := FALSE;
   PLI_AD[109] := FALSE;
   PLI_AD[110] := FALSE;
   PLI_AD[111] := FALSE;
   PLI_AD[112] := FALSE;
   PLI_AD[113] := FALSE;
   PLI_AD[114] := FALSE;
   PLI_AD[115] := FALSE;
   PLI_AD[116] := FALSE;
   PLI_AD[117] := FALSE;
   PLI_AD[118] := FALSE;
   PLI_AD[119] := FALSE;
   PLI_AD[120] := FALSE;
   PLI_AD[121] := FALSE;
   PLI_AD[122] := FALSE;
   PLI_AD[123] := FALSE;
   PLI_AD[124] := FALSE;
   PLI_AD[125] := FALSE;
   PLI_AD[126] := FALSE;
   PLI_AD[127] := FALSE;
   PLI_AD[128] := FALSE;
   PLI_AD[129] := FALSE;
   PLI_AD[130] := FALSE;
   PLI_AD[131] := FALSE;
   PLI_AD[132] := FALSE;
   PLI_AD[133] := FALSE;
   PLI_AD[134] := FALSE;
   PLI_AD[135] := FALSE;
   PLI_AD[136] := FALSE;
   PLI_AD[137] := FALSE;
   PLI_AD[138] := FALSE;
   PLI_AD[139] := FALSE;
   PLI_AD[140] := FALSE;
   PLI_AD[141] := FALSE;
   PLI_AD[142] := FALSE;
   PLI_AD[143] := FALSE;
   PLI_AD[144] := FALSE;
   PLI_AD[145] := FALSE;
   PLI_AD[146] := FALSE;
   PLI_AD[147] := FALSE;
   PLI_AD[148] := FALSE;
   PLI_AD[149] := FALSE;
   PLI_AD[150] := FALSE;
   PLI_HD[1] := FALSE;
   PLI_HD[2] := FALSE;
   PLI_HD[3] := FALSE;
   PLI_HD[4] := FALSE;
   PLI_HD[5] := FALSE;
   PLI_HD[6] := FALSE;
   PLI_HD[7] := FALSE;
   PLI_HD[8] := FALSE;
   PLI_HD[9] := FALSE;
   PLI_HD[10] := FALSE;
   PLI_HD[11] := FALSE;
   PLI_HD[12] := FALSE;
   PLI_HD[13] := FALSE;
   PLI_HD[14] := FALSE;
   PLI_HD[15] := FALSE;
   PLI_HD[16] := FALSE;
   PLI_HD[17] := FALSE;
   PLI_HD[18] := FALSE;
   PLI_HD[19] := FALSE;
   PLI_HD[20] := FALSE;
   PLI_HD[21] := FALSE;
   PLI_HD[22] := FALSE;
   PLI_HD[23] := FALSE;
   PLI_HD[24] := FALSE;
   PLI_HD[25] := FALSE;
   PLI_HD[26] := FALSE;
   PLI_HD[27] := FALSE;
   PLI_HD[28] := FALSE;
   PLI_HD[29] := FALSE;
   PLI_HD[30] := FALSE;
   PLI_HD[31] := FALSE;
   PLI_HD[32] := FALSE;
   PLI_HD[33] := FALSE;
   PLI_HD[34] := FALSE;
   PLI_HD[35] := FALSE;
   PLI_HD[36] := FALSE;
   PLI_HD[37] := FALSE;
   PLI_HD[38] := FALSE;
   PLI_HD[39] := FALSE;
   PLI_HD[40] := FALSE;
   PLI_HD[41] := FALSE;
   PLI_HD[42] := FALSE;
   PLI_HD[43] := FALSE;
   PLI_HD[44] := FALSE;
   PLI_HD[45] := FALSE;
   PLI_HD[46] := FALSE;
   PLI_HD[47] := FALSE;
   PLI_HD[48] := FALSE;
   PLI_HD[49] := FALSE;
   PLI_HD[50] := FALSE;
   PLI_HD[51] := FALSE;
   PLI_HD[52] := FALSE;
   PLI_HD[53] := FALSE;
   PLI_HD[54] := FALSE;
   PLI_HD[55] := FALSE;
   PLI_HD[56] := FALSE;
   PLI_HD[57] := FALSE;
   PLI_HD[58] := FALSE;
   PLI_HD[59] := FALSE;
   PLI_HD[60] := FALSE;
   PLI_HD[61] := FALSE;
   PLI_HD[62] := FALSE;
   PLI_HD[63] := FALSE;
   PLI_HD[64] := FALSE;
   PLI_HD[65] := FALSE;
   PLI_HD[66] := FALSE;
   PLI_HD[67] := FALSE;
   PLI_HD[68] := FALSE;
   PLI_HD[69] := FALSE;
   PLI_HD[70] := FALSE;
   PLI_HD[71] := FALSE;
   PLI_HD[72] := FALSE;
   PLI_HD[73] := TRUE;
   PLI_HD[74] := FALSE;
   PLI_HD[75] := FALSE;
   PLI_HD[76] := TRUE;
   PLI_HD[77] := FALSE;
   PLI_HD[78] := FALSE;
   PLI_HD[79] := FALSE;
   PLI_HD[80] := FALSE;
   PLI_HD[81] := FALSE;
   PLI_HD[82] := FALSE;
   PLI_HD[83] := FALSE;
   PLI_HD[84] := FALSE;
   PLI_HD[85] := FALSE;
   PLI_HD[86] := FALSE;
   PLI_HD[87] := FALSE;
   PLI_HD[88] := FALSE;
   PLI_HD[89] := FALSE;
   PLI_HD[90] := FALSE;
   PLI_HD[91] := FALSE;
   PLI_HD[92] := FALSE;
   PLI_HD[93] := FALSE;
   PLI_HD[94] := FALSE;
   PLI_HD[95] := FALSE;
   PLI_HD[96] := FALSE;
   PLI_HD[97] := FALSE;
   PLI_HD[98] := FALSE;
   PLI_HD[99] := FALSE;
   PLI_HD[100] := FALSE;
   PLI_HD[101] := FALSE;
   PLI_HD[102] := FALSE;
   PLI_HD[103] := FALSE;
   PLI_HD[104] := FALSE;
   PLI_HD[105] := FALSE;
   PLI_HD[106] := FALSE;
   PLI_HD[107] := FALSE;
   PLI_HD[108] := FALSE;
   PLI_HD[109] := FALSE;
   PLI_HD[110] := FALSE;
   PLI_HD[111] := FALSE;
   PLI_HD[112] := FALSE;
   PLI_HD[113] := FALSE;
   PLI_HD[114] := FALSE;
   PLI_HD[115] := FALSE;
   PLI_HD[116] := FALSE;
   PLI_HD[117] := FALSE;
   PLI_HD[118] := FALSE;
   PLI_HD[119] := FALSE;
   PLI_HD[120] := FALSE;
   PLI_HD[121] := FALSE;
   PLI_HD[122] := FALSE;
   PLI_HD[123] := FALSE;
   PLI_HD[124] := FALSE;
   PLI_HD[125] := FALSE;
   PLI_HD[126] := FALSE;
   PLI_HD[127] := FALSE;
   PLI_HD[128] := FALSE;
   PLI_HD[129] := FALSE;
   PLI_HD[130] := FALSE;
   PLI_HD[131] := FALSE;
   PLI_HD[132] := FALSE;
   PLI_HD[133] := FALSE;
   PLI_HD[134] := FALSE;
   PLI_HD[135] := FALSE;
   PLI_HD[136] := FALSE;
   PLI_HD[137] := FALSE;
   PLI_HD[138] := FALSE;
   PLI_HD[139] := FALSE;
   PLI_HD[140] := FALSE;
   PLI_HD[141] := FALSE;
   PLI_HD[142] := FALSE;
   PLI_HD[143] := FALSE;
   PLI_HD[144] := FALSE;
   PLI_HD[145] := FALSE;
   PLI_HD[146] := FALSE;
   PLI_HD[147] := FALSE;
   PLI_HD[148] := FALSE;
   PLI_HD[149] := FALSE;
   PLI_HD[150] := FALSE;
   PLI_SD[1] := FALSE;
   PLI_SD[2] := FALSE;
   PLI_SD[3] := FALSE;
   PLI_SD[4] := FALSE;
   PLI_SD[5] := FALSE;
   PLI_SD[6] := FALSE;
   PLI_SD[7] := FALSE;
   PLI_SD[8] := FALSE;
   PLI_SD[9] := FALSE;
   PLI_SD[10] := FALSE;
   PLI_SD[11] := FALSE;
   PLI_SD[12] := FALSE;
   PLI_SD[13] := FALSE;
   PLI_SD[14] := FALSE;
   PLI_SD[15] := FALSE;
   PLI_SD[16] := FALSE;
   PLI_SD[17] := FALSE;
   PLI_SD[18] := FALSE;
   PLI_SD[19] := FALSE;
   PLI_SD[20] := FALSE;
   PLI_SD[21] := FALSE;
   PLI_SD[22] := FALSE;
   PLI_SD[23] := FALSE;
   PLI_SD[24] := FALSE;
   PLI_SD[25] := FALSE;
   PLI_SD[26] := FALSE;
   PLI_SD[27] := FALSE;
   PLI_SD[28] := FALSE;
   PLI_SD[29] := FALSE;
   PLI_SD[30] := FALSE;
   PLI_SD[31] := FALSE;
   PLI_SD[32] := FALSE;
   PLI_SD[33] := FALSE;
   PLI_SD[34] := FALSE;
   PLI_SD[35] := FALSE;
   PLI_SD[36] := FALSE;
   PLI_SD[37] := FALSE;
   PLI_SD[38] := FALSE;
   PLI_SD[39] := FALSE;
   PLI_SD[40] := FALSE;
   PLI_SD[41] := FALSE;
   PLI_SD[42] := FALSE;
   PLI_SD[43] := FALSE;
   PLI_SD[44] := FALSE;
   PLI_SD[45] := FALSE;
   PLI_SD[46] := FALSE;
   PLI_SD[47] := FALSE;
   PLI_SD[48] := FALSE;
   PLI_SD[49] := FALSE;
   PLI_SD[50] := FALSE;
   PLI_SD[51] := FALSE;
   PLI_SD[52] := FALSE;
   PLI_SD[53] := FALSE;
   PLI_SD[54] := FALSE;
   PLI_SD[55] := FALSE;
   PLI_SD[56] := FALSE;
   PLI_SD[57] := FALSE;
   PLI_SD[58] := FALSE;
   PLI_SD[59] := FALSE;
   PLI_SD[60] := FALSE;
   PLI_SD[61] := FALSE;
   PLI_SD[62] := FALSE;
   PLI_SD[63] := FALSE;
   PLI_SD[64] := FALSE;
   PLI_SD[65] := FALSE;
   PLI_SD[66] := FALSE;
   PLI_SD[67] := FALSE;
   PLI_SD[68] := FALSE;
   PLI_SD[69] := FALSE;
   PLI_SD[70] := FALSE;
   PLI_SD[71] := FALSE;
   PLI_SD[72] := FALSE;
   PLI_SD[73] := FALSE;
   PLI_SD[74] := FALSE;
   PLI_SD[75] := FALSE;
   PLI_SD[76] := FALSE;
   PLI_SD[77] := FALSE;
   PLI_SD[78] := FALSE;
   PLI_SD[79] := FALSE;
   PLI_SD[80] := FALSE;
   PLI_SD[81] := FALSE;
   PLI_SD[82] := FALSE;
   PLI_SD[83] := FALSE;
   PLI_SD[84] := FALSE;
   PLI_SD[85] := FALSE;
   PLI_SD[86] := FALSE;
   PLI_SD[87] := FALSE;
   PLI_SD[88] := FALSE;
   PLI_SD[89] := FALSE;
   PLI_SD[90] := FALSE;
   PLI_SD[91] := FALSE;
   PLI_SD[92] := FALSE;
   PLI_SD[93] := FALSE;
   PLI_SD[94] := FALSE;
   PLI_SD[95] := FALSE;
   PLI_SD[96] := FALSE;
   PLI_SD[97] := FALSE;
   PLI_SD[98] := FALSE;
   PLI_SD[99] := FALSE;
   PLI_SD[100] := FALSE;
   PLI_SD[101] := FALSE;
   PLI_SD[102] := FALSE;
   PLI_SD[103] := FALSE;
   PLI_SD[104] := FALSE;
   PLI_SD[105] := FALSE;
   PLI_SD[106] := FALSE;
   PLI_SD[107] := FALSE;
   PLI_SD[108] := FALSE;
   PLI_SD[109] := FALSE;
   PLI_SD[110] := FALSE;
   PLI_SD[111] := FALSE;
   PLI_SD[112] := FALSE;
   PLI_SD[113] := FALSE;
   PLI_SD[114] := FALSE;
   PLI_SD[115] := FALSE;
   PLI_SD[116] := FALSE;
   PLI_SD[117] := FALSE;
   PLI_SD[118] := FALSE;
   PLI_SD[119] := FALSE;
   PLI_SD[120] := FALSE;
   PLI_SD[121] := FALSE;
   PLI_SD[122] := FALSE;
   PLI_SD[123] := FALSE;
   PLI_SD[124] := FALSE;
   PLI_SD[125] := FALSE;
   PLI_SD[126] := FALSE;
   PLI_SD[127] := FALSE;
   PLI_SD[128] := FALSE;
   PLI_SD[129] := FALSE;
   PLI_SD[130] := FALSE;
   PLI_SD[131] := FALSE;
   PLI_SD[132] := FALSE;
   PLI_SD[133] := FALSE;
   PLI_SD[134] := FALSE;
   PLI_SD[135] := FALSE;
   PLI_SD[136] := FALSE;
   PLI_SD[137] := FALSE;
   PLI_SD[138] := FALSE;
   PLI_SD[139] := FALSE;
   PLI_SD[140] := FALSE;
   PLI_SD[141] := FALSE;
   PLI_SD[142] := FALSE;
   PLI_SD[143] := FALSE;
   PLI_SD[144] := FALSE;
   PLI_SD[145] := FALSE;
   PLI_SD[146] := FALSE;
   PLI_SD[147] := FALSE;
   PLI_SD[148] := FALSE;
   PLI_SD[149] := FALSE;
   PLI_SD[150] := FALSE;
   PLI_FI[1] := FALSE;
   PLI_FI[2] := FALSE;
   PLI_FI[3] := FALSE;
   PLI_FI[4] := FALSE;
   PLI_FI[5] := FALSE;
   PLI_FI[6] := FALSE;
   PLI_FI[7] := FALSE;
   PLI_FI[8] := FALSE;
   PLI_FI[9] := FALSE;
   PLI_FI[10] := FALSE;
   PLI_FI[11] := FALSE;
   PLI_FI[12] := FALSE;
   PLI_FI[13] := FALSE;
   PLI_FI[14] := FALSE;
   PLI_FI[15] := FALSE;
   PLI_FI[16] := FALSE;
   PLI_FI[17] := FALSE;
   PLI_FI[18] := FALSE;
   PLI_FI[19] := FALSE;
   PLI_FI[20] := FALSE;
   PLI_FI[21] := FALSE;
   PLI_FI[22] := FALSE;
   PLI_FI[23] := FALSE;
   PLI_FI[24] := FALSE;
   PLI_FI[25] := FALSE;
   PLI_FI[26] := FALSE;
   PLI_FI[27] := FALSE;
   PLI_FI[28] := FALSE;
   PLI_FI[29] := FALSE;
   PLI_FI[30] := FALSE;
   PLI_FI[31] := FALSE;
   PLI_FI[32] := FALSE;
   PLI_FI[33] := FALSE;
   PLI_FI[34] := FALSE;
   PLI_FI[35] := FALSE;
   PLI_FI[36] := FALSE;
   PLI_FI[37] := FALSE;
   PLI_FI[38] := FALSE;
   PLI_FI[39] := FALSE;
   PLI_FI[40] := FALSE;
   PLI_FI[41] := FALSE;
   PLI_FI[42] := FALSE;
   PLI_FI[43] := FALSE;
   PLI_FI[44] := FALSE;
   PLI_FI[45] := FALSE;
   PLI_FI[46] := FALSE;
   PLI_FI[47] := FALSE;
   PLI_FI[48] := FALSE;
   PLI_FI[49] := FALSE;
   PLI_FI[50] := FALSE;
   PLI_FI[51] := FALSE;
   PLI_FI[52] := FALSE;
   PLI_FI[53] := FALSE;
   PLI_FI[54] := FALSE;
   PLI_FI[55] := FALSE;
   PLI_FI[56] := FALSE;
   PLI_FI[57] := FALSE;
   PLI_FI[58] := FALSE;
   PLI_FI[59] := FALSE;
   PLI_FI[60] := FALSE;
   PLI_FI[61] := FALSE;
   PLI_FI[62] := FALSE;
   PLI_FI[63] := FALSE;
   PLI_FI[64] := FALSE;
   PLI_FI[65] := FALSE;
   PLI_FI[66] := FALSE;
   PLI_FI[67] := FALSE;
   PLI_FI[68] := FALSE;
   PLI_FI[69] := FALSE;
   PLI_FI[70] := FALSE;
   PLI_FI[71] := FALSE;
   PLI_FI[72] := FALSE;
   PLI_FI[73] := FALSE;
   PLI_FI[74] := FALSE;
   PLI_FI[75] := FALSE;
   PLI_FI[76] := FALSE;
   PLI_FI[77] := FALSE;
   PLI_FI[78] := FALSE;
   PLI_FI[79] := FALSE;
   PLI_FI[80] := FALSE;
   PLI_FI[81] := FALSE;
   PLI_FI[82] := FALSE;
   PLI_FI[83] := FALSE;
   PLI_FI[84] := FALSE;
   PLI_FI[85] := FALSE;
   PLI_FI[86] := FALSE;
   PLI_FI[87] := FALSE;
   PLI_FI[88] := FALSE;
   PLI_FI[89] := FALSE;
   PLI_FI[90] := FALSE;
   PLI_FI[91] := FALSE;
   PLI_FI[92] := FALSE;
   PLI_FI[93] := FALSE;
   PLI_FI[94] := FALSE;
   PLI_FI[95] := FALSE;
   PLI_FI[96] := FALSE;
   PLI_FI[97] := FALSE;
   PLI_FI[98] := FALSE;
   PLI_FI[99] := FALSE;
   PLI_FI[100] := FALSE;
   PLI_FI[101] := FALSE;
   PLI_FI[102] := FALSE;
   PLI_FI[103] := FALSE;
   PLI_FI[104] := FALSE;
   PLI_FI[105] := FALSE;
   PLI_FI[106] := FALSE;
   PLI_FI[107] := FALSE;
   PLI_FI[108] := FALSE;
   PLI_FI[109] := FALSE;
   PLI_FI[110] := FALSE;
   PLI_FI[111] := FALSE;
   PLI_FI[112] := FALSE;
   PLI_FI[113] := FALSE;
   PLI_FI[114] := FALSE;
   PLI_FI[115] := FALSE;
   PLI_FI[116] := FALSE;
   PLI_FI[117] := FALSE;
   PLI_FI[118] := FALSE;
   PLI_FI[119] := FALSE;
   PLI_FI[120] := FALSE;
   PLI_FI[121] := FALSE;
   PLI_FI[122] := FALSE;
   PLI_FI[123] := FALSE;
   PLI_FI[124] := FALSE;
   PLI_FI[125] := FALSE;
   PLI_FI[126] := FALSE;
   PLI_FI[127] := FALSE;
   PLI_FI[128] := FALSE;
   PLI_FI[129] := FALSE;
   PLI_FI[130] := FALSE;
   PLI_FI[131] := FALSE;
   PLI_FI[132] := FALSE;
   PLI_FI[133] := FALSE;
   PLI_FI[134] := FALSE;
   PLI_FI[135] := FALSE;
   PLI_FI[136] := FALSE;
   PLI_FI[137] := FALSE;
   PLI_FI[138] := FALSE;
   PLI_FI[139] := FALSE;
   PLI_FI[140] := FALSE;
   PLI_FI[141] := FALSE;
   PLI_FI[142] := FALSE;
   PLI_FI[143] := FALSE;
   PLI_FI[144] := FALSE;
   PLI_FI[145] := FALSE;
   PLI_FI[146] := FALSE;
   PLI_FI[147] := FALSE;
   PLI_FI[148] := FALSE;
   PLI_FI[149] := FALSE;
   PLI_FI[150] := FALSE;
   PLI_W[1] := FALSE;
   PLI_W[2] := FALSE;
   PLI_W[3] := FALSE;
   PLI_W[4] := FALSE;
   PLI_W[5] := FALSE;
   PLI_W[6] := FALSE;
   PLI_W[7] := FALSE;
   PLI_W[8] := FALSE;
   PLI_W[9] := FALSE;
   PLI_W[10] := FALSE;
   PLI_W[11] := FALSE;
   PLI_W[12] := FALSE;
   PLI_W[13] := FALSE;
   PLI_W[14] := FALSE;
   PLI_W[15] := FALSE;
   PLI_W[16] := FALSE;
   PLI_W[17] := FALSE;
   PLI_W[18] := FALSE;
   PLI_W[19] := FALSE;
   PLI_W[20] := FALSE;
   PLI_W[21] := FALSE;
   PLI_W[22] := FALSE;
   PLI_W[23] := FALSE;
   PLI_W[24] := FALSE;
   PLI_W[25] := FALSE;
   PLI_W[26] := FALSE;
   PLI_W[27] := FALSE;
   PLI_W[28] := FALSE;
   PLI_W[29] := FALSE;
   PLI_W[30] := FALSE;
   PLI_W[31] := FALSE;
   PLI_W[32] := FALSE;
   PLI_W[33] := FALSE;
   PLI_W[34] := FALSE;
   PLI_W[35] := FALSE;
   PLI_W[36] := FALSE;
   PLI_W[37] := FALSE;
   PLI_W[38] := FALSE;
   PLI_W[39] := FALSE;
   PLI_W[40] := FALSE;
   PLI_W[41] := FALSE;
   PLI_W[42] := FALSE;
   PLI_W[43] := FALSE;
   PLI_W[44] := FALSE;
   PLI_W[45] := FALSE;
   PLI_W[46] := FALSE;
   PLI_W[47] := FALSE;
   PLI_W[48] := FALSE;
   PLI_W[49] := FALSE;
   PLI_W[50] := FALSE;
   PLI_W[51] := FALSE;
   PLI_W[52] := FALSE;
   PLI_W[53] := FALSE;
   PLI_W[54] := FALSE;
   PLI_W[55] := FALSE;
   PLI_W[56] := FALSE;
   PLI_W[57] := FALSE;
   PLI_W[58] := FALSE;
   PLI_W[59] := FALSE;
   PLI_W[60] := FALSE;
   PLI_W[61] := FALSE;
   PLI_W[62] := FALSE;
   PLI_W[63] := FALSE;
   PLI_W[64] := FALSE;
   PLI_W[65] := FALSE;
   PLI_W[66] := FALSE;
   PLI_W[67] := FALSE;
   PLI_W[68] := FALSE;
   PLI_W[69] := FALSE;
   PLI_W[70] := FALSE;
   PLI_W[71] := FALSE;
   PLI_W[72] := FALSE;
   PLI_W[73] := FALSE;
   PLI_W[74] := FALSE;
   PLI_W[75] := FALSE;
   PLI_W[76] := FALSE;
   PLI_W[77] := FALSE;
   PLI_W[78] := FALSE;
   PLI_W[79] := FALSE;
   PLI_W[80] := FALSE;
   PLI_W[81] := FALSE;
   PLI_W[82] := FALSE;
   PLI_W[83] := FALSE;
   PLI_W[84] := FALSE;
   PLI_W[85] := FALSE;
   PLI_W[86] := FALSE;
   PLI_W[87] := FALSE;
   PLI_W[88] := FALSE;
   PLI_W[89] := FALSE;
   PLI_W[90] := FALSE;
   PLI_W[91] := FALSE;
   PLI_W[92] := FALSE;
   PLI_W[93] := FALSE;
   PLI_W[94] := FALSE;
   PLI_W[95] := FALSE;
   PLI_W[96] := FALSE;
   PLI_W[97] := FALSE;
   PLI_W[98] := FALSE;
   PLI_W[99] := FALSE;
   PLI_W[100] := FALSE;
   PLI_W[101] := FALSE;
   PLI_W[102] := FALSE;
   PLI_W[103] := FALSE;
   PLI_W[104] := FALSE;
   PLI_W[105] := FALSE;
   PLI_W[106] := FALSE;
   PLI_W[107] := FALSE;
   PLI_W[108] := FALSE;
   PLI_W[109] := FALSE;
   PLI_W[110] := FALSE;
   PLI_W[111] := FALSE;
   PLI_W[112] := FALSE;
   PLI_W[113] := FALSE;
   PLI_W[114] := FALSE;
   PLI_W[115] := FALSE;
   PLI_W[116] := FALSE;
   PLI_W[117] := FALSE;
   PLI_W[118] := FALSE;
   PLI_W[119] := FALSE;
   PLI_W[120] := FALSE;
   PLI_W[121] := FALSE;
   PLI_W[122] := FALSE;
   PLI_W[123] := FALSE;
   PLI_W[124] := FALSE;
   PLI_W[125] := FALSE;
   PLI_W[126] := FALSE;
   PLI_W[127] := FALSE;
   PLI_W[128] := FALSE;
   PLI_W[129] := FALSE;
   PLI_W[130] := FALSE;
   PLI_W[131] := FALSE;
   PLI_W[132] := FALSE;
   PLI_W[133] := FALSE;
   PLI_W[134] := FALSE;
   PLI_W[135] := FALSE;
   PLI_W[136] := FALSE;
   PLI_W[137] := FALSE;
   PLI_W[138] := FALSE;
   PLI_W[139] := FALSE;
   PLI_W[140] := FALSE;
   PLI_W[141] := FALSE;
   PLI_W[142] := FALSE;
   PLI_W[143] := FALSE;
   PLI_W[144] := FALSE;
   PLI_W[145] := FALSE;
   PLI_W[146] := FALSE;
   PLI_W[147] := FALSE;
   PLI_W[148] := FALSE;
   PLI_W[149] := FALSE;
   PLI_W[150] := FALSE;
   PLI_P[1] := FALSE;
   PLI_P[2] := FALSE;
   PLI_P[3] := FALSE;
   PLI_P[4] := FALSE;
   PLI_P[5] := FALSE;
   PLI_P[6] := FALSE;
   PLI_P[7] := FALSE;
   PLI_P[8] := FALSE;
   PLI_P[9] := FALSE;
   PLI_P[10] := FALSE;
   PLI_P[11] := FALSE;
   PLI_P[12] := FALSE;
   PLI_P[13] := FALSE;
   PLI_P[14] := FALSE;
   PLI_P[15] := FALSE;
   PLI_P[16] := FALSE;
   PLI_P[17] := FALSE;
   PLI_P[18] := FALSE;
   PLI_P[19] := FALSE;
   PLI_P[20] := FALSE;
   PLI_P[21] := FALSE;
   PLI_P[22] := FALSE;
   PLI_P[23] := FALSE;
   PLI_P[24] := FALSE;
   PLI_P[25] := FALSE;
   PLI_P[26] := FALSE;
   PLI_P[27] := FALSE;
   PLI_P[28] := FALSE;
   PLI_P[29] := FALSE;
   PLI_P[30] := FALSE;
   PLI_P[31] := FALSE;
   PLI_P[32] := FALSE;
   PLI_P[33] := FALSE;
   PLI_P[34] := FALSE;
   PLI_P[35] := FALSE;
   PLI_P[36] := FALSE;
   PLI_P[37] := FALSE;
   PLI_P[38] := FALSE;
   PLI_P[39] := FALSE;
   PLI_P[40] := FALSE;
   PLI_P[41] := FALSE;
   PLI_P[42] := FALSE;
   PLI_P[43] := FALSE;
   PLI_P[44] := FALSE;
   PLI_P[45] := FALSE;
   PLI_P[46] := FALSE;
   PLI_P[47] := FALSE;
   PLI_P[48] := FALSE;
   PLI_P[49] := FALSE;
   PLI_P[50] := FALSE;
   PLI_P[51] := FALSE;
   PLI_P[52] := FALSE;
   PLI_P[53] := FALSE;
   PLI_P[54] := FALSE;
   PLI_P[55] := FALSE;
   PLI_P[56] := FALSE;
   PLI_P[57] := FALSE;
   PLI_P[58] := FALSE;
   PLI_P[59] := FALSE;
   PLI_P[60] := FALSE;
   PLI_P[61] := FALSE;
   PLI_P[62] := FALSE;
   PLI_P[63] := FALSE;
   PLI_P[64] := FALSE;
   PLI_P[65] := FALSE;
   PLI_P[66] := FALSE;
   PLI_P[67] := FALSE;
   PLI_P[68] := FALSE;
   PLI_P[69] := FALSE;
   PLI_P[70] := FALSE;
   PLI_P[71] := FALSE;
   PLI_P[72] := FALSE;
   PLI_P[73] := FALSE;
   PLI_P[74] := FALSE;
   PLI_P[75] := FALSE;
   PLI_P[76] := FALSE;
   PLI_P[77] := FALSE;
   PLI_P[78] := FALSE;
   PLI_P[79] := FALSE;
   PLI_P[80] := FALSE;
   PLI_P[81] := FALSE;
   PLI_P[82] := FALSE;
   PLI_P[83] := FALSE;
   PLI_P[84] := FALSE;
   PLI_P[85] := FALSE;
   PLI_P[86] := FALSE;
   PLI_P[87] := FALSE;
   PLI_P[88] := FALSE;
   PLI_P[89] := FALSE;
   PLI_P[90] := FALSE;
   PLI_P[91] := FALSE;
   PLI_P[92] := FALSE;
   PLI_P[93] := FALSE;
   PLI_P[94] := FALSE;
   PLI_P[95] := FALSE;
   PLI_P[96] := FALSE;
   PLI_P[97] := FALSE;
   PLI_P[98] := FALSE;
   PLI_P[99] := FALSE;
   PLI_P[100] := FALSE;
   PLI_P[101] := FALSE;
   PLI_P[102] := FALSE;
   PLI_P[103] := FALSE;
   PLI_P[104] := FALSE;
   PLI_P[105] := FALSE;
   PLI_P[106] := FALSE;
   PLI_P[107] := FALSE;
   PLI_P[108] := FALSE;
   PLI_P[109] := FALSE;
   PLI_P[110] := FALSE;
   PLI_P[111] := FALSE;
   PLI_P[112] := FALSE;
   PLI_P[113] := FALSE;
   PLI_P[114] := FALSE;
   PLI_P[115] := FALSE;
   PLI_P[116] := FALSE;
   PLI_P[117] := FALSE;
   PLI_P[118] := FALSE;
   PLI_P[119] := FALSE;
   PLI_P[120] := FALSE;
   PLI_P[121] := FALSE;
   PLI_P[122] := FALSE;
   PLI_P[123] := FALSE;
   PLI_P[124] := FALSE;
   PLI_P[125] := FALSE;
   PLI_P[126] := FALSE;
   PLI_P[127] := FALSE;
   PLI_P[128] := FALSE;
   PLI_P[129] := FALSE;
   PLI_P[130] := FALSE;
   PLI_P[131] := FALSE;
   PLI_P[132] := FALSE;
   PLI_P[133] := FALSE;
   PLI_P[134] := FALSE;
   PLI_P[135] := FALSE;
   PLI_P[136] := FALSE;
   PLI_P[137] := FALSE;
   PLI_P[138] := FALSE;
   PLI_P[139] := FALSE;
   PLI_P[140] := FALSE;
   PLI_P[141] := FALSE;
   PLI_P[142] := FALSE;
   PLI_P[143] := FALSE;
   PLI_P[144] := FALSE;
   PLI_P[145] := FALSE;
   PLI_P[146] := FALSE;
   PLI_P[147] := FALSE;
   PLI_P[148] := FALSE;
   PLI_P[149] := FALSE;
   PLI_P[150] := FALSE;
   PLI_PD[1] := FALSE;
   PLI_PD[2] := FALSE;
   PLI_PD[3] := FALSE;
   PLI_PD[4] := FALSE;
   PLI_PD[5] := FALSE;
   PLI_PD[6] := FALSE;
   PLI_PD[7] := FALSE;
   PLI_PD[8] := FALSE;
   PLI_PD[9] := FALSE;
   PLI_PD[10] := FALSE;
   PLI_PD[11] := FALSE;
   PLI_PD[12] := FALSE;
   PLI_PD[13] := FALSE;
   PLI_PD[14] := FALSE;
   PLI_PD[15] := FALSE;
   PLI_PD[16] := FALSE;
   PLI_PD[17] := FALSE;
   PLI_PD[18] := FALSE;
   PLI_PD[19] := FALSE;
   PLI_PD[20] := FALSE;
   PLI_PD[21] := FALSE;
   PLI_PD[22] := FALSE;
   PLI_PD[23] := FALSE;
   PLI_PD[24] := FALSE;
   PLI_PD[25] := FALSE;
   PLI_PD[26] := FALSE;
   PLI_PD[27] := FALSE;
   PLI_PD[28] := FALSE;
   PLI_PD[29] := FALSE;
   PLI_PD[30] := FALSE;
   PLI_PD[31] := FALSE;
   PLI_PD[32] := FALSE;
   PLI_PD[33] := FALSE;
   PLI_PD[34] := FALSE;
   PLI_PD[35] := FALSE;
   PLI_PD[36] := FALSE;
   PLI_PD[37] := FALSE;
   PLI_PD[38] := FALSE;
   PLI_PD[39] := FALSE;
   PLI_PD[40] := FALSE;
   PLI_PD[41] := FALSE;
   PLI_PD[42] := FALSE;
   PLI_PD[43] := FALSE;
   PLI_PD[44] := FALSE;
   PLI_PD[45] := FALSE;
   PLI_PD[46] := FALSE;
   PLI_PD[47] := FALSE;
   PLI_PD[48] := FALSE;
   PLI_PD[49] := FALSE;
   PLI_PD[50] := FALSE;
   PLI_PD[51] := FALSE;
   PLI_PD[52] := FALSE;
   PLI_PD[53] := FALSE;
   PLI_PD[54] := FALSE;
   PLI_PD[55] := FALSE;
   PLI_PD[56] := FALSE;
   PLI_PD[57] := FALSE;
   PLI_PD[58] := FALSE;
   PLI_PD[59] := FALSE;
   PLI_PD[60] := FALSE;
   PLI_PD[61] := FALSE;
   PLI_PD[62] := FALSE;
   PLI_PD[63] := FALSE;
   PLI_PD[64] := FALSE;
   PLI_PD[65] := FALSE;
   PLI_PD[66] := FALSE;
   PLI_PD[67] := FALSE;
   PLI_PD[68] := FALSE;
   PLI_PD[69] := FALSE;
   PLI_PD[70] := FALSE;
   PLI_PD[71] := FALSE;
   PLI_PD[72] := FALSE;
   PLI_PD[73] := FALSE;
   PLI_PD[74] := FALSE;
   PLI_PD[75] := FALSE;
   PLI_PD[76] := FALSE;
   PLI_PD[77] := FALSE;
   PLI_PD[78] := FALSE;
   PLI_PD[79] := FALSE;
   PLI_PD[80] := FALSE;
   PLI_PD[81] := FALSE;
   PLI_PD[82] := FALSE;
   PLI_PD[83] := FALSE;
   PLI_PD[84] := FALSE;
   PLI_PD[85] := FALSE;
   PLI_PD[86] := FALSE;
   PLI_PD[87] := FALSE;
   PLI_PD[88] := FALSE;
   PLI_PD[89] := FALSE;
   PLI_PD[90] := FALSE;
   PLI_PD[91] := FALSE;
   PLI_PD[92] := FALSE;
   PLI_PD[93] := FALSE;
   PLI_PD[94] := FALSE;
   PLI_PD[95] := FALSE;
   PLI_PD[96] := FALSE;
   PLI_PD[97] := FALSE;
   PLI_PD[98] := FALSE;
   PLI_PD[99] := FALSE;
   PLI_PD[100] := FALSE;
   PLI_PD[101] := FALSE;
   PLI_PD[102] := FALSE;
   PLI_PD[103] := FALSE;
   PLI_PD[104] := FALSE;
   PLI_PD[105] := FALSE;
   PLI_PD[106] := FALSE;
   PLI_PD[107] := FALSE;
   PLI_PD[108] := FALSE;
   PLI_PD[109] := FALSE;
   PLI_PD[110] := FALSE;
   PLI_PD[111] := FALSE;
   PLI_PD[112] := FALSE;
   PLI_PD[113] := FALSE;
   PLI_PD[114] := FALSE;
   PLI_PD[115] := FALSE;
   PLI_PD[116] := FALSE;
   PLI_PD[117] := FALSE;
   PLI_PD[118] := FALSE;
   PLI_PD[119] := FALSE;
   PLI_PD[120] := FALSE;
   PLI_PD[121] := FALSE;
   PLI_PD[122] := FALSE;
   PLI_PD[123] := FALSE;
   PLI_PD[124] := FALSE;
   PLI_PD[125] := FALSE;
   PLI_PD[126] := FALSE;
   PLI_PD[127] := FALSE;
   PLI_PD[128] := FALSE;
   PLI_PD[129] := FALSE;
   PLI_PD[130] := FALSE;
   PLI_PD[131] := FALSE;
   PLI_PD[132] := FALSE;
   PLI_PD[133] := FALSE;
   PLI_PD[134] := FALSE;
   PLI_PD[135] := FALSE;
   PLI_PD[136] := FALSE;
   PLI_PD[137] := FALSE;
   PLI_PD[138] := FALSE;
   PLI_PD[139] := FALSE;
   PLI_PD[140] := FALSE;
   PLI_PD[141] := FALSE;
   PLI_PD[142] := FALSE;
   PLI_PD[143] := FALSE;
   PLI_PD[144] := FALSE;
   PLI_PD[145] := FALSE;
   PLI_PD[146] := FALSE;
   PLI_PD[147] := FALSE;
   PLI_PD[148] := FALSE;
   PLI_PD[149] := FALSE;
   PLI_PD[150] := FALSE;
   PLI_SS[1] := FALSE;
   PLI_SS[2] := FALSE;
   PLI_SS[3] := FALSE;
   PLI_SS[4] := FALSE;
   PLI_SS[5] := FALSE;
   PLI_SS[6] := FALSE;
   PLI_SS[7] := FALSE;
   PLI_SS[8] := FALSE;
   PLI_SS[9] := FALSE;
   PLI_SS[10] := FALSE;
   PLI_SS[11] := FALSE;
   PLI_SS[12] := FALSE;
   PLI_SS[13] := FALSE;
   PLI_SS[14] := FALSE;
   PLI_SS[15] := FALSE;
   PLI_SS[16] := FALSE;
   PLI_SS[17] := FALSE;
   PLI_SS[18] := FALSE;
   PLI_SS[19] := FALSE;
   PLI_SS[20] := FALSE;
   PLI_SS[21] := FALSE;
   PLI_SS[22] := FALSE;
   PLI_SS[23] := FALSE;
   PLI_SS[24] := FALSE;
   PLI_SS[25] := FALSE;
   PLI_SS[26] := FALSE;
   PLI_SS[27] := FALSE;
   PLI_SS[28] := FALSE;
   PLI_SS[29] := FALSE;
   PLI_SS[30] := FALSE;
   PLI_SS[31] := FALSE;
   PLI_SS[32] := FALSE;
   PLI_SS[33] := FALSE;
   PLI_SS[34] := FALSE;
   PLI_SS[35] := FALSE;
   PLI_SS[36] := FALSE;
   PLI_SS[37] := FALSE;
   PLI_SS[38] := FALSE;
   PLI_SS[39] := FALSE;
   PLI_SS[40] := FALSE;
   PLI_SS[41] := FALSE;
   PLI_SS[42] := FALSE;
   PLI_SS[43] := FALSE;
   PLI_SS[44] := FALSE;
   PLI_SS[45] := FALSE;
   PLI_SS[46] := FALSE;
   PLI_SS[47] := FALSE;
   PLI_SS[48] := FALSE;
   PLI_SS[49] := FALSE;
   PLI_SS[50] := FALSE;
   PLI_SS[51] := FALSE;
   PLI_SS[52] := FALSE;
   PLI_SS[53] := FALSE;
   PLI_SS[54] := FALSE;
   PLI_SS[55] := FALSE;
   PLI_SS[56] := FALSE;
   PLI_SS[57] := FALSE;
   PLI_SS[58] := FALSE;
   PLI_SS[59] := FALSE;
   PLI_SS[60] := FALSE;
   PLI_SS[61] := FALSE;
   PLI_SS[62] := FALSE;
   PLI_SS[63] := FALSE;
   PLI_SS[64] := FALSE;
   PLI_SS[65] := FALSE;
   PLI_SS[66] := FALSE;
   PLI_SS[67] := FALSE;
   PLI_SS[68] := FALSE;
   PLI_SS[69] := FALSE;
   PLI_SS[70] := FALSE;
   PLI_SS[71] := FALSE;
   PLI_SS[72] := FALSE;
   PLI_SS[73] := FALSE;
   PLI_SS[74] := FALSE;
   PLI_SS[75] := FALSE;
   PLI_SS[76] := FALSE;
   PLI_SS[77] := FALSE;
   PLI_SS[78] := FALSE;
   PLI_SS[79] := FALSE;
   PLI_SS[80] := FALSE;
   PLI_SS[81] := FALSE;
   PLI_SS[82] := FALSE;
   PLI_SS[83] := FALSE;
   PLI_SS[84] := FALSE;
   PLI_SS[85] := FALSE;
   PLI_SS[86] := FALSE;
   PLI_SS[87] := FALSE;
   PLI_SS[88] := FALSE;
   PLI_SS[89] := FALSE;
   PLI_SS[90] := FALSE;
   PLI_SS[91] := FALSE;
   PLI_SS[92] := FALSE;
   PLI_SS[93] := FALSE;
   PLI_SS[94] := FALSE;
   PLI_SS[95] := FALSE;
   PLI_SS[96] := FALSE;
   PLI_SS[97] := FALSE;
   PLI_SS[98] := FALSE;
   PLI_SS[99] := FALSE;
   PLI_SS[100] := FALSE;
   PLI_SS[101] := FALSE;
   PLI_SS[102] := FALSE;
   PLI_SS[103] := FALSE;
   PLI_SS[104] := FALSE;
   PLI_SS[105] := FALSE;
   PLI_SS[106] := FALSE;
   PLI_SS[107] := FALSE;
   PLI_SS[108] := FALSE;
   PLI_SS[109] := FALSE;
   PLI_SS[110] := FALSE;
   PLI_SS[111] := FALSE;
   PLI_SS[112] := FALSE;
   PLI_SS[113] := FALSE;
   PLI_SS[114] := FALSE;
   PLI_SS[115] := FALSE;
   PLI_SS[116] := FALSE;
   PLI_SS[117] := FALSE;
   PLI_SS[118] := FALSE;
   PLI_SS[119] := FALSE;
   PLI_SS[120] := FALSE;
   PLI_SS[121] := FALSE;
   PLI_SS[122] := FALSE;
   PLI_SS[123] := FALSE;
   PLI_SS[124] := FALSE;
   PLI_SS[125] := FALSE;
   PLI_SS[126] := FALSE;
   PLI_SS[127] := FALSE;
   PLI_SS[128] := FALSE;
   PLI_SS[129] := FALSE;
   PLI_SS[130] := FALSE;
   PLI_SS[131] := FALSE;
   PLI_SS[132] := FALSE;
   PLI_SS[133] := FALSE;
   PLI_SS[134] := FALSE;
   PLI_SS[135] := FALSE;
   PLI_SS[136] := FALSE;
   PLI_SS[137] := FALSE;
   PLI_SS[138] := FALSE;
   PLI_SS[139] := FALSE;
   PLI_SS[140] := FALSE;
   PLI_SS[141] := FALSE;
   PLI_SS[142] := FALSE;
   PLI_SS[143] := FALSE;
   PLI_SS[144] := FALSE;
   PLI_SS[145] := FALSE;
   PLI_SS[146] := FALSE;
   PLI_SS[147] := FALSE;
   PLI_SS[148] := FALSE;
   PLI_SS[149] := FALSE;
   PLI_SS[150] := FALSE;
   PLI_NC[1] := FALSE;
   PLI_NC[2] := FALSE;
   PLI_NC[3] := FALSE;
   PLI_NC[4] := FALSE;
   PLI_NC[5] := FALSE;
   PLI_NC[6] := FALSE;
   PLI_NC[7] := FALSE;
   PLI_NC[8] := FALSE;
   PLI_NC[9] := FALSE;
   PLI_NC[10] := FALSE;
   PLI_NC[11] := FALSE;
   PLI_NC[12] := FALSE;
   PLI_NC[13] := FALSE;
   PLI_NC[14] := FALSE;
   PLI_NC[15] := FALSE;
   PLI_NC[16] := FALSE;
   PLI_NC[17] := FALSE;
   PLI_NC[18] := FALSE;
   PLI_NC[19] := FALSE;
   PLI_NC[20] := FALSE;
   PLI_NC[21] := FALSE;
   PLI_NC[22] := FALSE;
   PLI_NC[23] := FALSE;
   PLI_NC[24] := FALSE;
   PLI_NC[25] := FALSE;
   PLI_NC[26] := FALSE;
   PLI_NC[27] := FALSE;
   PLI_NC[28] := FALSE;
   PLI_NC[29] := FALSE;
   PLI_NC[30] := FALSE;
   PLI_NC[31] := FALSE;
   PLI_NC[32] := FALSE;
   PLI_NC[33] := FALSE;
   PLI_NC[34] := FALSE;
   PLI_NC[35] := FALSE;
   PLI_NC[36] := FALSE;
   PLI_NC[37] := FALSE;
   PLI_NC[38] := FALSE;
   PLI_NC[39] := FALSE;
   PLI_NC[40] := FALSE;
   PLI_NC[41] := FALSE;
   PLI_NC[42] := FALSE;
   PLI_NC[43] := FALSE;
   PLI_NC[44] := FALSE;
   PLI_NC[45] := FALSE;
   PLI_NC[46] := FALSE;
   PLI_NC[47] := FALSE;
   PLI_NC[48] := FALSE;
   PLI_NC[49] := FALSE;
   PLI_NC[50] := FALSE;
   PLI_NC[51] := FALSE;
   PLI_NC[52] := FALSE;
   PLI_NC[53] := FALSE;
   PLI_NC[54] := FALSE;
   PLI_NC[55] := FALSE;
   PLI_NC[56] := FALSE;
   PLI_NC[57] := FALSE;
   PLI_NC[58] := FALSE;
   PLI_NC[59] := FALSE;
   PLI_NC[60] := FALSE;
   PLI_NC[61] := FALSE;
   PLI_NC[62] := FALSE;
   PLI_NC[63] := FALSE;
   PLI_NC[64] := FALSE;
   PLI_NC[65] := FALSE;
   PLI_NC[66] := FALSE;
   PLI_NC[67] := FALSE;
   PLI_NC[68] := FALSE;
   PLI_NC[69] := FALSE;
   PLI_NC[70] := FALSE;
   PLI_NC[71] := FALSE;
   PLI_NC[72] := FALSE;
   PLI_NC[73] := FALSE;
   PLI_NC[74] := FALSE;
   PLI_NC[75] := FALSE;
   PLI_NC[76] := FALSE;
   PLI_NC[77] := FALSE;
   PLI_NC[78] := FALSE;
   PLI_NC[79] := FALSE;
   PLI_NC[80] := FALSE;
   PLI_NC[81] := FALSE;
   PLI_NC[82] := FALSE;
   PLI_NC[83] := FALSE;
   PLI_NC[84] := FALSE;
   PLI_NC[85] := FALSE;
   PLI_NC[86] := FALSE;
   PLI_NC[87] := FALSE;
   PLI_NC[88] := FALSE;
   PLI_NC[89] := FALSE;
   PLI_NC[90] := FALSE;
   PLI_NC[91] := FALSE;
   PLI_NC[92] := FALSE;
   PLI_NC[93] := FALSE;
   PLI_NC[94] := FALSE;
   PLI_NC[95] := FALSE;
   PLI_NC[96] := FALSE;
   PLI_NC[97] := FALSE;
   PLI_NC[98] := FALSE;
   PLI_NC[99] := FALSE;
   PLI_NC[100] := FALSE;
   PLI_NC[101] := FALSE;
   PLI_NC[102] := FALSE;
   PLI_NC[103] := FALSE;
   PLI_NC[104] := FALSE;
   PLI_NC[105] := FALSE;
   PLI_NC[106] := FALSE;
   PLI_NC[107] := FALSE;
   PLI_NC[108] := FALSE;
   PLI_NC[109] := FALSE;
   PLI_NC[110] := FALSE;
   PLI_NC[111] := FALSE;
   PLI_NC[112] := FALSE;
   PLI_NC[113] := FALSE;
   PLI_NC[114] := FALSE;
   PLI_NC[115] := FALSE;
   PLI_NC[116] := FALSE;
   PLI_NC[117] := FALSE;
   PLI_NC[118] := FALSE;
   PLI_NC[119] := FALSE;
   PLI_NC[120] := FALSE;
   PLI_NC[121] := FALSE;
   PLI_NC[122] := FALSE;
   PLI_NC[123] := FALSE;
   PLI_NC[124] := FALSE;
   PLI_NC[125] := FALSE;
   PLI_NC[126] := FALSE;
   PLI_NC[127] := FALSE;
   PLI_NC[128] := FALSE;
   PLI_NC[129] := FALSE;
   PLI_NC[130] := FALSE;
   PLI_NC[131] := FALSE;
   PLI_NC[132] := FALSE;
   PLI_NC[133] := FALSE;
   PLI_NC[134] := FALSE;
   PLI_NC[135] := FALSE;
   PLI_NC[136] := FALSE;
   PLI_NC[137] := FALSE;
   PLI_NC[138] := FALSE;
   PLI_NC[139] := FALSE;
   PLI_NC[140] := FALSE;
   PLI_NC[141] := FALSE;
   PLI_NC[142] := FALSE;
   PLI_NC[143] := FALSE;
   PLI_NC[144] := FALSE;
   PLI_NC[145] := FALSE;
   PLI_NC[146] := FALSE;
   PLI_NC[147] := FALSE;
   PLI_NC[148] := FALSE;
   PLI_NC[149] := FALSE;
   PLI_NC[150] := FALSE;
   PLI_IN[1] := FALSE;
   PLI_IN[2] := FALSE;
   PLI_IN[3] := FALSE;
   PLI_IN[4] := FALSE;
   PLI_IN[5] := FALSE;
   PLI_IN[6] := FALSE;
   PLI_IN[7] := FALSE;
   PLI_IN[8] := FALSE;
   PLI_IN[9] := FALSE;
   PLI_IN[10] := FALSE;
   PLI_IN[11] := FALSE;
   PLI_IN[12] := FALSE;
   PLI_IN[13] := FALSE;
   PLI_IN[14] := FALSE;
   PLI_IN[15] := FALSE;
   PLI_IN[16] := FALSE;
   PLI_IN[17] := FALSE;
   PLI_IN[18] := FALSE;
   PLI_IN[19] := FALSE;
   PLI_IN[20] := FALSE;
   PLI_IN[21] := FALSE;
   PLI_IN[22] := FALSE;
   PLI_IN[23] := FALSE;
   PLI_IN[24] := FALSE;
   PLI_IN[25] := FALSE;
   PLI_IN[26] := FALSE;
   PLI_IN[27] := FALSE;
   PLI_IN[28] := FALSE;
   PLI_IN[29] := FALSE;
   PLI_IN[30] := FALSE;
   PLI_IN[31] := FALSE;
   PLI_IN[32] := FALSE;
   PLI_IN[33] := FALSE;
   PLI_IN[34] := FALSE;
   PLI_IN[35] := FALSE;
   PLI_IN[36] := FALSE;
   PLI_IN[37] := FALSE;
   PLI_IN[38] := FALSE;
   PLI_IN[39] := FALSE;
   PLI_IN[40] := FALSE;
   PLI_IN[41] := FALSE;
   PLI_IN[42] := FALSE;
   PLI_IN[43] := FALSE;
   PLI_IN[44] := FALSE;
   PLI_IN[45] := FALSE;
   PLI_IN[46] := FALSE;
   PLI_IN[47] := FALSE;
   PLI_IN[48] := FALSE;
   PLI_IN[49] := FALSE;
   PLI_IN[50] := FALSE;
   PLI_IN[51] := FALSE;
   PLI_IN[52] := FALSE;
   PLI_IN[53] := FALSE;
   PLI_IN[54] := FALSE;
   PLI_IN[55] := FALSE;
   PLI_IN[56] := FALSE;
   PLI_IN[57] := FALSE;
   PLI_IN[58] := FALSE;
   PLI_IN[59] := FALSE;
   PLI_IN[60] := FALSE;
   PLI_IN[61] := FALSE;
   PLI_IN[62] := FALSE;
   PLI_IN[63] := FALSE;
   PLI_IN[64] := FALSE;
   PLI_IN[65] := FALSE;
   PLI_IN[66] := FALSE;
   PLI_IN[67] := FALSE;
   PLI_IN[68] := FALSE;
   PLI_IN[69] := FALSE;
   PLI_IN[70] := FALSE;
   PLI_IN[71] := FALSE;
   PLI_IN[72] := FALSE;
   PLI_IN[73] := FALSE;
   PLI_IN[74] := FALSE;
   PLI_IN[75] := FALSE;
   PLI_IN[76] := FALSE;
   PLI_IN[77] := FALSE;
   PLI_IN[78] := FALSE;
   PLI_IN[79] := FALSE;
   PLI_IN[80] := FALSE;
   PLI_IN[81] := FALSE;
   PLI_IN[82] := FALSE;
   PLI_IN[83] := FALSE;
   PLI_IN[84] := FALSE;
   PLI_IN[85] := FALSE;
   PLI_IN[86] := FALSE;
   PLI_IN[87] := FALSE;
   PLI_IN[88] := FALSE;
   PLI_IN[89] := FALSE;
   PLI_IN[90] := FALSE;
   PLI_IN[91] := FALSE;
   PLI_IN[92] := FALSE;
   PLI_IN[93] := FALSE;
   PLI_IN[94] := FALSE;
   PLI_IN[95] := FALSE;
   PLI_IN[96] := FALSE;
   PLI_IN[97] := FALSE;
   PLI_IN[98] := FALSE;
   PLI_IN[99] := FALSE;
   PLI_IN[100] := FALSE;
   PLI_IN[101] := FALSE;
   PLI_IN[102] := FALSE;
   PLI_IN[103] := FALSE;
   PLI_IN[104] := FALSE;
   PLI_IN[105] := FALSE;
   PLI_IN[106] := FALSE;
   PLI_IN[107] := FALSE;
   PLI_IN[108] := FALSE;
   PLI_IN[109] := FALSE;
   PLI_IN[110] := FALSE;
   PLI_IN[111] := FALSE;
   PLI_IN[112] := FALSE;
   PLI_IN[113] := FALSE;
   PLI_IN[114] := FALSE;
   PLI_IN[115] := FALSE;
   PLI_IN[116] := FALSE;
   PLI_IN[117] := FALSE;
   PLI_IN[118] := FALSE;
   PLI_IN[119] := FALSE;
   PLI_IN[120] := FALSE;
   PLI_IN[121] := FALSE;
   PLI_IN[122] := FALSE;
   PLI_IN[123] := FALSE;
   PLI_IN[124] := FALSE;
   PLI_IN[125] := FALSE;
   PLI_IN[126] := FALSE;
   PLI_IN[127] := FALSE;
   PLI_IN[128] := FALSE;
   PLI_IN[129] := FALSE;
   PLI_IN[130] := FALSE;
   PLI_IN[131] := FALSE;
   PLI_IN[132] := FALSE;
   PLI_IN[133] := FALSE;
   PLI_IN[134] := FALSE;
   PLI_IN[135] := FALSE;
   PLI_IN[136] := FALSE;
   PLI_IN[137] := FALSE;
   PLI_IN[138] := FALSE;
   PLI_IN[139] := FALSE;
   PLI_IN[140] := FALSE;
   PLI_IN[141] := FALSE;
   PLI_IN[142] := FALSE;
   PLI_IN[143] := FALSE;
   PLI_IN[144] := FALSE;
   PLI_IN[145] := FALSE;
   PLI_IN[146] := FALSE;
   PLI_IN[147] := FALSE;
   PLI_IN[148] := FALSE;
   PLI_IN[149] := FALSE;
   PLI_IN[150] := FALSE;
   PLI_ER[1] := FALSE;
   PLI_ER[2] := FALSE;
   PLI_ER[3] := FALSE;
   PLI_ER[4] := FALSE;
   PLI_ER[5] := FALSE;
   PLI_ER[6] := FALSE;
   PLI_ER[7] := FALSE;
   PLI_ER[8] := FALSE;
   PLI_ER[9] := FALSE;
   PLI_ER[10] := FALSE;
   PLI_ER[11] := FALSE;
   PLI_ER[12] := FALSE;
   PLI_ER[13] := FALSE;
   PLI_ER[14] := FALSE;
   PLI_ER[15] := FALSE;
   PLI_ER[16] := FALSE;
   PLI_ER[17] := FALSE;
   PLI_ER[18] := FALSE;
   PLI_ER[19] := FALSE;
   PLI_ER[20] := FALSE;
   PLI_ER[21] := FALSE;
   PLI_ER[22] := FALSE;
   PLI_ER[23] := FALSE;
   PLI_ER[24] := FALSE;
   PLI_ER[25] := FALSE;
   PLI_ER[26] := FALSE;
   PLI_ER[27] := FALSE;
   PLI_ER[28] := FALSE;
   PLI_ER[29] := FALSE;
   PLI_ER[30] := FALSE;
   PLI_ER[31] := FALSE;
   PLI_ER[32] := FALSE;
   PLI_ER[33] := FALSE;
   PLI_ER[34] := FALSE;
   PLI_ER[35] := FALSE;
   PLI_ER[36] := FALSE;
   PLI_ER[37] := FALSE;
   PLI_ER[38] := FALSE;
   PLI_ER[39] := FALSE;
   PLI_ER[40] := FALSE;
   PLI_ER[41] := FALSE;
   PLI_ER[42] := FALSE;
   PLI_ER[43] := FALSE;
   PLI_ER[44] := FALSE;
   PLI_ER[45] := FALSE;
   PLI_ER[46] := FALSE;
   PLI_ER[47] := FALSE;
   PLI_ER[48] := FALSE;
   PLI_ER[49] := FALSE;
   PLI_ER[50] := FALSE;
   PLI_ER[51] := FALSE;
   PLI_ER[52] := FALSE;
   PLI_ER[53] := FALSE;
   PLI_ER[54] := FALSE;
   PLI_ER[55] := FALSE;
   PLI_ER[56] := FALSE;
   PLI_ER[57] := FALSE;
   PLI_ER[58] := FALSE;
   PLI_ER[59] := FALSE;
   PLI_ER[60] := FALSE;
   PLI_ER[61] := FALSE;
   PLI_ER[62] := FALSE;
   PLI_ER[63] := FALSE;
   PLI_ER[64] := FALSE;
   PLI_ER[65] := FALSE;
   PLI_ER[66] := FALSE;
   PLI_ER[67] := FALSE;
   PLI_ER[68] := FALSE;
   PLI_ER[69] := FALSE;
   PLI_ER[70] := FALSE;
   PLI_ER[71] := FALSE;
   PLI_ER[72] := FALSE;
   PLI_ER[73] := FALSE;
   PLI_ER[74] := FALSE;
   PLI_ER[75] := FALSE;
   PLI_ER[76] := FALSE;
   PLI_ER[77] := FALSE;
   PLI_ER[78] := FALSE;
   PLI_ER[79] := FALSE;
   PLI_ER[80] := FALSE;
   PLI_ER[81] := FALSE;
   PLI_ER[82] := FALSE;
   PLI_ER[83] := FALSE;
   PLI_ER[84] := FALSE;
   PLI_ER[85] := FALSE;
   PLI_ER[86] := FALSE;
   PLI_ER[87] := FALSE;
   PLI_ER[88] := FALSE;
   PLI_ER[89] := FALSE;
   PLI_ER[90] := FALSE;
   PLI_ER[91] := FALSE;
   PLI_ER[92] := FALSE;
   PLI_ER[93] := FALSE;
   PLI_ER[94] := FALSE;
   PLI_ER[95] := FALSE;
   PLI_ER[96] := FALSE;
   PLI_ER[97] := FALSE;
   PLI_ER[98] := FALSE;
   PLI_ER[99] := FALSE;
   PLI_ER[100] := FALSE;
   PLI_ER[101] := FALSE;
   PLI_ER[102] := FALSE;
   PLI_ER[103] := FALSE;
   PLI_ER[104] := FALSE;
   PLI_ER[105] := FALSE;
   PLI_ER[106] := FALSE;
   PLI_ER[107] := FALSE;
   PLI_ER[108] := FALSE;
   PLI_ER[109] := FALSE;
   PLI_ER[110] := FALSE;
   PLI_ER[111] := FALSE;
   PLI_ER[112] := FALSE;
   PLI_ER[113] := FALSE;
   PLI_ER[114] := FALSE;
   PLI_ER[115] := FALSE;
   PLI_ER[116] := FALSE;
   PLI_ER[117] := FALSE;
   PLI_ER[118] := FALSE;
   PLI_ER[119] := FALSE;
   PLI_ER[120] := FALSE;
   PLI_ER[121] := FALSE;
   PLI_ER[122] := FALSE;
   PLI_ER[123] := FALSE;
   PLI_ER[124] := FALSE;
   PLI_ER[125] := FALSE;
   PLI_ER[126] := FALSE;
   PLI_ER[127] := FALSE;
   PLI_ER[128] := FALSE;
   PLI_ER[129] := FALSE;
   PLI_ER[130] := FALSE;
   PLI_ER[131] := FALSE;
   PLI_ER[132] := FALSE;
   PLI_ER[133] := FALSE;
   PLI_ER[134] := FALSE;
   PLI_ER[135] := FALSE;
   PLI_ER[136] := FALSE;
   PLI_ER[137] := FALSE;
   PLI_ER[138] := FALSE;
   PLI_ER[139] := FALSE;
   PLI_ER[140] := FALSE;
   PLI_ER[141] := FALSE;
   PLI_ER[142] := FALSE;
   PLI_ER[143] := FALSE;
   PLI_ER[144] := FALSE;
   PLI_ER[145] := FALSE;
   PLI_ER[146] := FALSE;
   PLI_ER[147] := FALSE;
   PLI_ER[148] := FALSE;
   PLI_ER[149] := FALSE;
   PLI_ER[150] := FALSE;
   PLI_OR[1] := FALSE;
   PLI_OR[2] := FALSE;
   PLI_OR[3] := FALSE;
   PLI_OR[4] := FALSE;
   PLI_OR[5] := FALSE;
   PLI_OR[6] := FALSE;
   PLI_OR[7] := FALSE;
   PLI_OR[8] := FALSE;
   PLI_OR[9] := FALSE;
   PLI_OR[10] := FALSE;
   PLI_OR[11] := FALSE;
   PLI_OR[12] := FALSE;
   PLI_OR[13] := FALSE;
   PLI_OR[14] := FALSE;
   PLI_OR[15] := FALSE;
   PLI_OR[16] := FALSE;
   PLI_OR[17] := FALSE;
   PLI_OR[18] := FALSE;
   PLI_OR[19] := FALSE;
   PLI_OR[20] := FALSE;
   PLI_OR[21] := FALSE;
   PLI_OR[22] := FALSE;
   PLI_OR[23] := FALSE;
   PLI_OR[24] := FALSE;
   PLI_OR[25] := FALSE;
   PLI_OR[26] := FALSE;
   PLI_OR[27] := FALSE;
   PLI_OR[28] := FALSE;
   PLI_OR[29] := FALSE;
   PLI_OR[30] := FALSE;
   PLI_OR[31] := FALSE;
   PLI_OR[32] := FALSE;
   PLI_OR[33] := FALSE;
   PLI_OR[34] := FALSE;
   PLI_OR[35] := FALSE;
   PLI_OR[36] := FALSE;
   PLI_OR[37] := FALSE;
   PLI_OR[38] := FALSE;
   PLI_OR[39] := FALSE;
   PLI_OR[40] := FALSE;
   PLI_OR[41] := FALSE;
   PLI_OR[42] := FALSE;
   PLI_OR[43] := FALSE;
   PLI_OR[44] := FALSE;
   PLI_OR[45] := FALSE;
   PLI_OR[46] := FALSE;
   PLI_OR[47] := FALSE;
   PLI_OR[48] := FALSE;
   PLI_OR[49] := FALSE;
   PLI_OR[50] := FALSE;
   PLI_OR[51] := FALSE;
   PLI_OR[52] := FALSE;
   PLI_OR[53] := FALSE;
   PLI_OR[54] := FALSE;
   PLI_OR[55] := FALSE;
   PLI_OR[56] := FALSE;
   PLI_OR[57] := FALSE;
   PLI_OR[58] := FALSE;
   PLI_OR[59] := FALSE;
   PLI_OR[60] := FALSE;
   PLI_OR[61] := FALSE;
   PLI_OR[62] := FALSE;
   PLI_OR[63] := FALSE;
   PLI_OR[64] := FALSE;
   PLI_OR[65] := FALSE;
   PLI_OR[66] := FALSE;
   PLI_OR[67] := FALSE;
   PLI_OR[68] := FALSE;
   PLI_OR[69] := FALSE;
   PLI_OR[70] := FALSE;
   PLI_OR[71] := FALSE;
   PLI_OR[72] := FALSE;
   PLI_OR[73] := FALSE;
   PLI_OR[74] := FALSE;
   PLI_OR[75] := FALSE;
   PLI_OR[76] := FALSE;
   PLI_OR[77] := FALSE;
   PLI_OR[78] := FALSE;
   PLI_OR[79] := FALSE;
   PLI_OR[80] := FALSE;
   PLI_OR[81] := FALSE;
   PLI_OR[82] := FALSE;
   PLI_OR[83] := FALSE;
   PLI_OR[84] := FALSE;
   PLI_OR[85] := FALSE;
   PLI_OR[86] := FALSE;
   PLI_OR[87] := FALSE;
   PLI_OR[88] := FALSE;
   PLI_OR[89] := FALSE;
   PLI_OR[90] := FALSE;
   PLI_OR[91] := FALSE;
   PLI_OR[92] := FALSE;
   PLI_OR[93] := FALSE;
   PLI_OR[94] := FALSE;
   PLI_OR[95] := FALSE;
   PLI_OR[96] := FALSE;
   PLI_OR[97] := FALSE;
   PLI_OR[98] := FALSE;
   PLI_OR[99] := FALSE;
   PLI_OR[100] := FALSE;
   PLI_OR[101] := FALSE;
   PLI_OR[102] := FALSE;
   PLI_OR[103] := FALSE;
   PLI_OR[104] := FALSE;
   PLI_OR[105] := FALSE;
   PLI_OR[106] := FALSE;
   PLI_OR[107] := FALSE;
   PLI_OR[108] := FALSE;
   PLI_OR[109] := FALSE;
   PLI_OR[110] := FALSE;
   PLI_OR[111] := FALSE;
   PLI_OR[112] := FALSE;
   PLI_OR[113] := FALSE;
   PLI_OR[114] := FALSE;
   PLI_OR[115] := FALSE;
   PLI_OR[116] := FALSE;
   PLI_OR[117] := FALSE;
   PLI_OR[118] := FALSE;
   PLI_OR[119] := FALSE;
   PLI_OR[120] := FALSE;
   PLI_OR[121] := FALSE;
   PLI_OR[122] := FALSE;
   PLI_OR[123] := FALSE;
   PLI_OR[124] := FALSE;
   PLI_OR[125] := FALSE;
   PLI_OR[126] := FALSE;
   PLI_OR[127] := FALSE;
   PLI_OR[128] := FALSE;
   PLI_OR[129] := FALSE;
   PLI_OR[130] := FALSE;
   PLI_OR[131] := FALSE;
   PLI_OR[132] := FALSE;
   PLI_OR[133] := FALSE;
   PLI_OR[134] := FALSE;
   PLI_OR[135] := FALSE;
   PLI_OR[136] := FALSE;
   PLI_OR[137] := FALSE;
   PLI_OR[138] := FALSE;
   PLI_OR[139] := FALSE;
   PLI_OR[140] := FALSE;
   PLI_OR[141] := FALSE;
   PLI_OR[142] := FALSE;
   PLI_OR[143] := FALSE;
   PLI_OR[144] := FALSE;
   PLI_OR[145] := FALSE;
   PLI_OR[146] := FALSE;
   PLI_OR[147] := FALSE;
   PLI_OR[148] := FALSE;
   PLI_OR[149] := FALSE;
   PLI_OR[150] := FALSE;
   PLI_RR[1] := FALSE;
   PLI_RR[2] := FALSE;
   PLI_RR[3] := FALSE;
   PLI_RR[4] := FALSE;
   PLI_RR[5] := FALSE;
   PLI_RR[6] := FALSE;
   PLI_RR[7] := FALSE;
   PLI_RR[8] := FALSE;
   PLI_RR[9] := FALSE;
   PLI_RR[10] := FALSE;
   PLI_RR[11] := FALSE;
   PLI_RR[12] := FALSE;
   PLI_RR[13] := FALSE;
   PLI_RR[14] := FALSE;
   PLI_RR[15] := FALSE;
   PLI_RR[16] := FALSE;
   PLI_RR[17] := FALSE;
   PLI_RR[18] := FALSE;
   PLI_RR[19] := FALSE;
   PLI_RR[20] := FALSE;
   PLI_RR[21] := FALSE;
   PLI_RR[22] := FALSE;
   PLI_RR[23] := FALSE;
   PLI_RR[24] := FALSE;
   PLI_RR[25] := FALSE;
   PLI_RR[26] := FALSE;
   PLI_RR[27] := FALSE;
   PLI_RR[28] := FALSE;
   PLI_RR[29] := FALSE;
   PLI_RR[30] := FALSE;
   PLI_RR[31] := FALSE;
   PLI_RR[32] := FALSE;
   PLI_RR[33] := FALSE;
   PLI_RR[34] := FALSE;
   PLI_RR[35] := FALSE;
   PLI_RR[36] := FALSE;
   PLI_RR[37] := FALSE;
   PLI_RR[38] := FALSE;
   PLI_RR[39] := FALSE;
   PLI_RR[40] := FALSE;
   PLI_RR[41] := FALSE;
   PLI_RR[42] := FALSE;
   PLI_RR[43] := FALSE;
   PLI_RR[44] := FALSE;
   PLI_RR[45] := FALSE;
   PLI_RR[46] := FALSE;
   PLI_RR[47] := FALSE;
   PLI_RR[48] := FALSE;
   PLI_RR[49] := FALSE;
   PLI_RR[50] := FALSE;
   PLI_RR[51] := FALSE;
   PLI_RR[52] := FALSE;
   PLI_RR[53] := FALSE;
   PLI_RR[54] := FALSE;
   PLI_RR[55] := FALSE;
   PLI_RR[56] := FALSE;
   PLI_RR[57] := FALSE;
   PLI_RR[58] := FALSE;
   PLI_RR[59] := FALSE;
   PLI_RR[60] := FALSE;
   PLI_RR[61] := FALSE;
   PLI_RR[62] := FALSE;
   PLI_RR[63] := FALSE;
   PLI_RR[64] := FALSE;
   PLI_RR[65] := FALSE;
   PLI_RR[66] := FALSE;
   PLI_RR[67] := FALSE;
   PLI_RR[68] := FALSE;
   PLI_RR[69] := FALSE;
   PLI_RR[70] := FALSE;
   PLI_RR[71] := FALSE;
   PLI_RR[72] := FALSE;
   PLI_RR[73] := FALSE;
   PLI_RR[74] := FALSE;
   PLI_RR[75] := FALSE;
   PLI_RR[76] := FALSE;
   PLI_RR[77] := FALSE;
   PLI_RR[78] := FALSE;
   PLI_RR[79] := FALSE;
   PLI_RR[80] := FALSE;
   PLI_RR[81] := FALSE;
   PLI_RR[82] := FALSE;
   PLI_RR[83] := FALSE;
   PLI_RR[84] := FALSE;
   PLI_RR[85] := FALSE;
   PLI_RR[86] := FALSE;
   PLI_RR[87] := FALSE;
   PLI_RR[88] := FALSE;
   PLI_RR[89] := FALSE;
   PLI_RR[90] := FALSE;
   PLI_RR[91] := FALSE;
   PLI_RR[92] := FALSE;
   PLI_RR[93] := FALSE;
   PLI_RR[94] := FALSE;
   PLI_RR[95] := FALSE;
   PLI_RR[96] := FALSE;
   PLI_RR[97] := FALSE;
   PLI_RR[98] := FALSE;
   PLI_RR[99] := FALSE;
   PLI_RR[100] := FALSE;
   PLI_RR[101] := FALSE;
   PLI_RR[102] := FALSE;
   PLI_RR[103] := FALSE;
   PLI_RR[104] := FALSE;
   PLI_RR[105] := FALSE;
   PLI_RR[106] := FALSE;
   PLI_RR[107] := FALSE;
   PLI_RR[108] := FALSE;
   PLI_RR[109] := FALSE;
   PLI_RR[110] := FALSE;
   PLI_RR[111] := FALSE;
   PLI_RR[112] := FALSE;
   PLI_RR[113] := FALSE;
   PLI_RR[114] := FALSE;
   PLI_RR[115] := FALSE;
   PLI_RR[116] := FALSE;
   PLI_RR[117] := FALSE;
   PLI_RR[118] := FALSE;
   PLI_RR[119] := FALSE;
   PLI_RR[120] := FALSE;
   PLI_RR[121] := FALSE;
   PLI_RR[122] := FALSE;
   PLI_RR[123] := FALSE;
   PLI_RR[124] := FALSE;
   PLI_RR[125] := FALSE;
   PLI_RR[126] := FALSE;
   PLI_RR[127] := FALSE;
   PLI_RR[128] := FALSE;
   PLI_RR[129] := FALSE;
   PLI_RR[130] := FALSE;
   PLI_RR[131] := FALSE;
   PLI_RR[132] := FALSE;
   PLI_RR[133] := FALSE;
   PLI_RR[134] := FALSE;
   PLI_RR[135] := FALSE;
   PLI_RR[136] := FALSE;
   PLI_RR[137] := FALSE;
   PLI_RR[138] := FALSE;
   PLI_RR[139] := FALSE;
   PLI_RR[140] := FALSE;
   PLI_RR[141] := FALSE;
   PLI_RR[142] := FALSE;
   PLI_RR[143] := FALSE;
   PLI_RR[144] := FALSE;
   PLI_RR[145] := FALSE;
   PLI_RR[146] := FALSE;
   PLI_RR[147] := FALSE;
   PLI_RR[148] := FALSE;
   PLI_RR[149] := FALSE;
   PLI_RR[150] := FALSE;
   PLI_CR[1] := TRUE;
   PLI_CR[2] := TRUE;
   PLI_CR[3] := TRUE;
   PLI_CR[4] := TRUE;
   PLI_CR[5] := TRUE;
   PLI_CR[6] := TRUE;
   PLI_CR[7] := TRUE;
   PLI_CR[8] := TRUE;
   PLI_CR[9] := TRUE;
   PLI_CR[10] := TRUE;
   PLI_CR[11] := TRUE;
   PLI_CR[12] := TRUE;
   PLI_CR[13] := TRUE;
   PLI_CR[14] := TRUE;
   PLI_CR[15] := TRUE;
   PLI_CR[16] := TRUE;
   PLI_CR[17] := TRUE;
   PLI_CR[18] := TRUE;
   PLI_CR[19] := TRUE;
   PLI_CR[20] := TRUE;
   PLI_CR[21] := TRUE;
   PLI_CR[22] := TRUE;
   PLI_CR[23] := TRUE;
   PLI_CR[24] := TRUE;
   PLI_CR[25] := TRUE;
   PLI_CR[26] := TRUE;
   PLI_CR[27] := TRUE;
   PLI_CR[28] := TRUE;
   PLI_CR[29] := TRUE;
   PLI_CR[30] := TRUE;
   PLI_CR[31] := TRUE;
   PLI_CR[32] := TRUE;
   PLI_CR[33] := TRUE;
   PLI_CR[34] := TRUE;
   PLI_CR[35] := TRUE;
   PLI_CR[36] := TRUE;
   PLI_CR[37] := TRUE;
   PLI_CR[38] := TRUE;
   PLI_CR[39] := TRUE;
   PLI_CR[40] := TRUE;
   PLI_CR[41] := TRUE;
   PLI_CR[42] := TRUE;
   PLI_CR[43] := TRUE;
   PLI_CR[44] := TRUE;
   PLI_CR[45] := TRUE;
   PLI_CR[46] := TRUE;
   PLI_CR[47] := TRUE;
   PLI_CR[48] := TRUE;
   PLI_CR[49] := TRUE;
   PLI_CR[50] := TRUE;
   PLI_CR[51] := TRUE;
   PLI_CR[52] := TRUE;
   PLI_CR[53] := TRUE;
   PLI_CR[54] := TRUE;
   PLI_CR[55] := TRUE;
   PLI_CR[56] := TRUE;
   PLI_CR[57] := TRUE;
   PLI_CR[58] := TRUE;
   PLI_CR[59] := TRUE;
   PLI_CR[60] := TRUE;
   PLI_CR[61] := TRUE;
   PLI_CR[62] := TRUE;
   PLI_CR[63] := TRUE;
   PLI_CR[64] := TRUE;
   PLI_CR[65] := TRUE;
   PLI_CR[66] := TRUE;
   PLI_CR[67] := TRUE;
   PLI_CR[68] := TRUE;
   PLI_CR[69] := TRUE;
   PLI_CR[70] := TRUE;
   PLI_CR[71] := TRUE;
   PLI_CR[72] := TRUE;
   PLI_CR[73] := TRUE;
   PLI_CR[74] := TRUE;
   PLI_CR[75] := TRUE;
   PLI_CR[76] := TRUE;
   PLI_CR[77] := TRUE;
   PLI_CR[78] := TRUE;
   PLI_CR[79] := TRUE;
   PLI_CR[80] := TRUE;
   PLI_CR[81] := TRUE;
   PLI_CR[82] := TRUE;
   PLI_CR[83] := TRUE;
   PLI_CR[84] := TRUE;
   PLI_CR[85] := TRUE;
   PLI_CR[86] := TRUE;
   PLI_CR[87] := TRUE;
   PLI_CR[88] := TRUE;
   PLI_CR[89] := TRUE;
   PLI_CR[90] := TRUE;
   PLI_CR[91] := TRUE;
   PLI_CR[92] := TRUE;
   PLI_CR[93] := TRUE;
   PLI_CR[94] := TRUE;
   PLI_CR[95] := TRUE;
   PLI_CR[96] := TRUE;
   PLI_CR[97] := TRUE;
   PLI_CR[98] := TRUE;
   PLI_CR[99] := TRUE;
   PLI_CR[100] := TRUE;
   PLI_CR[101] := TRUE;
   PLI_CR[102] := TRUE;
   PLI_CR[103] := TRUE;
   PLI_CR[104] := TRUE;
   PLI_CR[105] := TRUE;
   PLI_CR[106] := TRUE;
   PLI_CR[107] := TRUE;
   PLI_CR[108] := TRUE;
   PLI_CR[109] := TRUE;
   PLI_CR[110] := TRUE;
   PLI_CR[111] := TRUE;
   PLI_CR[112] := TRUE;
   PLI_CR[113] := TRUE;
   PLI_CR[114] := TRUE;
   PLI_CR[115] := TRUE;
   PLI_CR[116] := TRUE;
   PLI_CR[117] := TRUE;
   PLI_CR[118] := TRUE;
   PLI_CR[119] := TRUE;
   PLI_CR[120] := TRUE;
   PLI_CR[121] := TRUE;
   PLI_CR[122] := TRUE;
   PLI_CR[123] := TRUE;
   PLI_CR[124] := TRUE;
   PLI_CR[125] := TRUE;
   PLI_CR[126] := TRUE;
   PLI_CR[127] := TRUE;
   PLI_CR[128] := TRUE;
   PLI_CR[129] := TRUE;
   PLI_CR[130] := TRUE;
   PLI_CR[131] := TRUE;
   PLI_CR[132] := TRUE;
   PLI_CR[133] := TRUE;
   PLI_CR[134] := TRUE;
   PLI_CR[135] := TRUE;
   PLI_CR[136] := TRUE;
   PLI_CR[137] := TRUE;
   PLI_CR[138] := TRUE;
   PLI_CR[139] := TRUE;
   PLI_CR[140] := TRUE;
   PLI_CR[141] := TRUE;
   PLI_CR[142] := TRUE;
   PLI_CR[143] := TRUE;
   PLI_CR[144] := TRUE;
   PLI_CR[145] := TRUE;
   PLI_CR[146] := TRUE;
   PLI_CR[147] := TRUE;
   PLI_CR[148] := TRUE;
   PLI_CR[149] := TRUE;
   PLI_CR[150] := TRUE;
   PLI_RE[1] := FALSE;
   PLI_RE[2] := FALSE;
   PLI_RE[3] := FALSE;
   PLI_RE[4] := FALSE;
   PLI_RE[5] := FALSE;
   PLI_RE[6] := FALSE;
   PLI_RE[7] := FALSE;
   PLI_RE[8] := FALSE;
   PLI_RE[9] := FALSE;
   PLI_RE[10] := FALSE;
   PLI_RE[11] := FALSE;
   PLI_RE[12] := FALSE;
   PLI_RE[13] := FALSE;
   PLI_RE[14] := FALSE;
   PLI_RE[15] := FALSE;
   PLI_RE[16] := FALSE;
   PLI_RE[17] := FALSE;
   PLI_RE[18] := FALSE;
   PLI_RE[19] := FALSE;
   PLI_RE[20] := FALSE;
   PLI_RE[21] := FALSE;
   PLI_RE[22] := FALSE;
   PLI_RE[23] := FALSE;
   PLI_RE[24] := FALSE;
   PLI_RE[25] := FALSE;
   PLI_RE[26] := FALSE;
   PLI_RE[27] := FALSE;
   PLI_RE[28] := FALSE;
   PLI_RE[29] := FALSE;
   PLI_RE[30] := FALSE;
   PLI_RE[31] := FALSE;
   PLI_RE[32] := FALSE;
   PLI_RE[33] := FALSE;
   PLI_RE[34] := FALSE;
   PLI_RE[35] := FALSE;
   PLI_RE[36] := FALSE;
   PLI_RE[37] := FALSE;
   PLI_RE[38] := FALSE;
   PLI_RE[39] := FALSE;
   PLI_RE[40] := FALSE;
   PLI_RE[41] := FALSE;
   PLI_RE[42] := FALSE;
   PLI_RE[43] := FALSE;
   PLI_RE[44] := FALSE;
   PLI_RE[45] := FALSE;
   PLI_RE[46] := FALSE;
   PLI_RE[47] := FALSE;
   PLI_RE[48] := FALSE;
   PLI_RE[49] := FALSE;
   PLI_RE[50] := FALSE;
   PLI_RE[51] := FALSE;
   PLI_RE[52] := FALSE;
   PLI_RE[53] := FALSE;
   PLI_RE[54] := FALSE;
   PLI_RE[55] := FALSE;
   PLI_RE[56] := FALSE;
   PLI_RE[57] := FALSE;
   PLI_RE[58] := FALSE;
   PLI_RE[59] := FALSE;
   PLI_RE[60] := FALSE;
   PLI_RE[61] := FALSE;
   PLI_RE[62] := FALSE;
   PLI_RE[63] := FALSE;
   PLI_RE[64] := FALSE;
   PLI_RE[65] := FALSE;
   PLI_RE[66] := FALSE;
   PLI_RE[67] := FALSE;
   PLI_RE[68] := FALSE;
   PLI_RE[69] := FALSE;
   PLI_RE[70] := FALSE;
   PLI_RE[71] := FALSE;
   PLI_RE[72] := FALSE;
   PLI_RE[73] := FALSE;
   PLI_RE[74] := FALSE;
   PLI_RE[75] := FALSE;
   PLI_RE[76] := FALSE;
   PLI_RE[77] := FALSE;
   PLI_RE[78] := FALSE;
   PLI_RE[79] := FALSE;
   PLI_RE[80] := FALSE;
   PLI_RE[81] := FALSE;
   PLI_RE[82] := FALSE;
   PLI_RE[83] := FALSE;
   PLI_RE[84] := FALSE;
   PLI_RE[85] := FALSE;
   PLI_RE[86] := FALSE;
   PLI_RE[87] := FALSE;
   PLI_RE[88] := FALSE;
   PLI_RE[89] := FALSE;
   PLI_RE[90] := FALSE;
   PLI_RE[91] := FALSE;
   PLI_RE[92] := FALSE;
   PLI_RE[93] := FALSE;
   PLI_RE[94] := FALSE;
   PLI_RE[95] := FALSE;
   PLI_RE[96] := FALSE;
   PLI_RE[97] := FALSE;
   PLI_RE[98] := FALSE;
   PLI_RE[99] := FALSE;
   PLI_RE[100] := FALSE;
   PLI_RE[101] := FALSE;
   PLI_RE[102] := FALSE;
   PLI_RE[103] := FALSE;
   PLI_RE[104] := FALSE;
   PLI_RE[105] := FALSE;
   PLI_RE[106] := FALSE;
   PLI_RE[107] := FALSE;
   PLI_RE[108] := FALSE;
   PLI_RE[109] := FALSE;
   PLI_RE[110] := FALSE;
   PLI_RE[111] := FALSE;
   PLI_RE[112] := FALSE;
   PLI_RE[113] := FALSE;
   PLI_RE[114] := FALSE;
   PLI_RE[115] := FALSE;
   PLI_RE[116] := FALSE;
   PLI_RE[117] := FALSE;
   PLI_RE[118] := FALSE;
   PLI_RE[119] := FALSE;
   PLI_RE[120] := FALSE;
   PLI_RE[121] := FALSE;
   PLI_RE[122] := FALSE;
   PLI_RE[123] := FALSE;
   PLI_RE[124] := FALSE;
   PLI_RE[125] := FALSE;
   PLI_RE[126] := FALSE;
   PLI_RE[127] := FALSE;
   PLI_RE[128] := FALSE;
   PLI_RE[129] := FALSE;
   PLI_RE[130] := FALSE;
   PLI_RE[131] := FALSE;
   PLI_RE[132] := FALSE;
   PLI_RE[133] := FALSE;
   PLI_RE[134] := FALSE;
   PLI_RE[135] := FALSE;
   PLI_RE[136] := FALSE;
   PLI_RE[137] := FALSE;
   PLI_RE[138] := FALSE;
   PLI_RE[139] := FALSE;
   PLI_RE[140] := FALSE;
   PLI_RE[141] := FALSE;
   PLI_RE[142] := FALSE;
   PLI_RE[143] := FALSE;
   PLI_RE[144] := FALSE;
   PLI_RE[145] := FALSE;
   PLI_RE[146] := FALSE;
   PLI_RE[147] := FALSE;
   PLI_RE[148] := FALSE;
   PLI_RE[149] := FALSE;
   PLI_RE[150] := FALSE;
   PLI_DL[1] := FALSE;
   PLI_DL[2] := FALSE;
   PLI_DL[3] := FALSE;
   PLI_DL[4] := FALSE;
   PLI_DL[5] := FALSE;
   PLI_DL[6] := FALSE;
   PLI_DL[7] := FALSE;
   PLI_DL[8] := FALSE;
   PLI_DL[9] := FALSE;
   PLI_DL[10] := FALSE;
   PLI_DL[11] := FALSE;
   PLI_DL[12] := FALSE;
   PLI_DL[13] := FALSE;
   PLI_DL[14] := FALSE;
   PLI_DL[15] := FALSE;
   PLI_DL[16] := FALSE;
   PLI_DL[17] := FALSE;
   PLI_DL[18] := FALSE;
   PLI_DL[19] := FALSE;
   PLI_DL[20] := FALSE;
   PLI_DL[21] := FALSE;
   PLI_DL[22] := FALSE;
   PLI_DL[23] := FALSE;
   PLI_DL[24] := FALSE;
   PLI_DL[25] := FALSE;
   PLI_DL[26] := FALSE;
   PLI_DL[27] := FALSE;
   PLI_DL[28] := FALSE;
   PLI_DL[29] := FALSE;
   PLI_DL[30] := FALSE;
   PLI_DL[31] := FALSE;
   PLI_DL[32] := FALSE;
   PLI_DL[33] := FALSE;
   PLI_DL[34] := FALSE;
   PLI_DL[35] := FALSE;
   PLI_DL[36] := FALSE;
   PLI_DL[37] := FALSE;
   PLI_DL[38] := FALSE;
   PLI_DL[39] := FALSE;
   PLI_DL[40] := FALSE;
   PLI_DL[41] := FALSE;
   PLI_DL[42] := FALSE;
   PLI_DL[43] := FALSE;
   PLI_DL[44] := FALSE;
   PLI_DL[45] := FALSE;
   PLI_DL[46] := FALSE;
   PLI_DL[47] := FALSE;
   PLI_DL[48] := FALSE;
   PLI_DL[49] := FALSE;
   PLI_DL[50] := FALSE;
   PLI_DL[51] := FALSE;
   PLI_DL[52] := FALSE;
   PLI_DL[53] := FALSE;
   PLI_DL[54] := FALSE;
   PLI_DL[55] := FALSE;
   PLI_DL[56] := FALSE;
   PLI_DL[57] := FALSE;
   PLI_DL[58] := FALSE;
   PLI_DL[59] := FALSE;
   PLI_DL[60] := FALSE;
   PLI_DL[61] := FALSE;
   PLI_DL[62] := FALSE;
   PLI_DL[63] := FALSE;
   PLI_DL[64] := FALSE;
   PLI_DL[65] := FALSE;
   PLI_DL[66] := FALSE;
   PLI_DL[67] := FALSE;
   PLI_DL[68] := FALSE;
   PLI_DL[69] := FALSE;
   PLI_DL[70] := FALSE;
   PLI_DL[71] := FALSE;
   PLI_DL[72] := FALSE;
   PLI_DL[73] := FALSE;
   PLI_DL[74] := FALSE;
   PLI_DL[75] := FALSE;
   PLI_DL[76] := FALSE;
   PLI_DL[77] := FALSE;
   PLI_DL[78] := FALSE;
   PLI_DL[79] := FALSE;
   PLI_DL[80] := FALSE;
   PLI_DL[81] := FALSE;
   PLI_DL[82] := FALSE;
   PLI_DL[83] := FALSE;
   PLI_DL[84] := FALSE;
   PLI_DL[85] := FALSE;
   PLI_DL[86] := FALSE;
   PLI_DL[87] := FALSE;
   PLI_DL[88] := FALSE;
   PLI_DL[89] := FALSE;
   PLI_DL[90] := FALSE;
   PLI_DL[91] := FALSE;
   PLI_DL[92] := FALSE;
   PLI_DL[93] := FALSE;
   PLI_DL[94] := FALSE;
   PLI_DL[95] := FALSE;
   PLI_DL[96] := FALSE;
   PLI_DL[97] := FALSE;
   PLI_DL[98] := FALSE;
   PLI_DL[99] := FALSE;
   PLI_DL[100] := FALSE;
   PLI_DL[101] := FALSE;
   PLI_DL[102] := FALSE;
   PLI_DL[103] := FALSE;
   PLI_DL[104] := FALSE;
   PLI_DL[105] := FALSE;
   PLI_DL[106] := FALSE;
   PLI_DL[107] := FALSE;
   PLI_DL[108] := FALSE;
   PLI_DL[109] := FALSE;
   PLI_DL[110] := FALSE;
   PLI_DL[111] := FALSE;
   PLI_DL[112] := FALSE;
   PLI_DL[113] := FALSE;
   PLI_DL[114] := FALSE;
   PLI_DL[115] := FALSE;
   PLI_DL[116] := FALSE;
   PLI_DL[117] := FALSE;
   PLI_DL[118] := FALSE;
   PLI_DL[119] := FALSE;
   PLI_DL[120] := FALSE;
   PLI_DL[121] := FALSE;
   PLI_DL[122] := FALSE;
   PLI_DL[123] := FALSE;
   PLI_DL[124] := FALSE;
   PLI_DL[125] := FALSE;
   PLI_DL[126] := FALSE;
   PLI_DL[127] := FALSE;
   PLI_DL[128] := FALSE;
   PLI_DL[129] := FALSE;
   PLI_DL[130] := FALSE;
   PLI_DL[131] := FALSE;
   PLI_DL[132] := FALSE;
   PLI_DL[133] := FALSE;
   PLI_DL[134] := FALSE;
   PLI_DL[135] := FALSE;
   PLI_DL[136] := FALSE;
   PLI_DL[137] := FALSE;
   PLI_DL[138] := FALSE;
   PLI_DL[139] := FALSE;
   PLI_DL[140] := FALSE;
   PLI_DL[141] := FALSE;
   PLI_DL[142] := FALSE;
   PLI_DL[143] := FALSE;
   PLI_DL[144] := FALSE;
   PLI_DL[145] := FALSE;
   PLI_DL[146] := FALSE;
   PLI_DL[147] := FALSE;
   PLI_DL[148] := FALSE;
   PLI_DL[149] := FALSE;
   PLI_DL[150] := FALSE;
   PLI_WC[1] := FALSE;
   PLI_WC[2] := FALSE;
   PLI_WC[3] := FALSE;
   PLI_WC[4] := FALSE;
   PLI_WC[5] := FALSE;
   PLI_WC[6] := FALSE;
   PLI_WC[7] := FALSE;
   PLI_WC[8] := FALSE;
   PLI_WC[9] := FALSE;
   PLI_WC[10] := FALSE;
   PLI_WC[11] := FALSE;
   PLI_WC[12] := FALSE;
   PLI_WC[13] := FALSE;
   PLI_WC[14] := FALSE;
   PLI_WC[15] := FALSE;
   PLI_WC[16] := FALSE;
   PLI_WC[17] := FALSE;
   PLI_WC[18] := FALSE;
   PLI_WC[19] := FALSE;
   PLI_WC[20] := FALSE;
   PLI_WC[21] := FALSE;
   PLI_WC[22] := FALSE;
   PLI_WC[23] := FALSE;
   PLI_WC[24] := FALSE;
   PLI_WC[25] := FALSE;
   PLI_WC[26] := FALSE;
   PLI_WC[27] := FALSE;
   PLI_WC[28] := FALSE;
   PLI_WC[29] := FALSE;
   PLI_WC[30] := FALSE;
   PLI_WC[31] := FALSE;
   PLI_WC[32] := FALSE;
   PLI_WC[33] := FALSE;
   PLI_WC[34] := FALSE;
   PLI_WC[35] := FALSE;
   PLI_WC[36] := FALSE;
   PLI_WC[37] := FALSE;
   PLI_WC[38] := FALSE;
   PLI_WC[39] := FALSE;
   PLI_WC[40] := FALSE;
   PLI_WC[41] := FALSE;
   PLI_WC[42] := FALSE;
   PLI_WC[43] := FALSE;
   PLI_WC[44] := FALSE;
   PLI_WC[45] := FALSE;
   PLI_WC[46] := FALSE;
   PLI_WC[47] := FALSE;
   PLI_WC[48] := FALSE;
   PLI_WC[49] := FALSE;
   PLI_WC[50] := FALSE;
   PLI_WC[51] := FALSE;
   PLI_WC[52] := FALSE;
   PLI_WC[53] := FALSE;
   PLI_WC[54] := FALSE;
   PLI_WC[55] := FALSE;
   PLI_WC[56] := FALSE;
   PLI_WC[57] := FALSE;
   PLI_WC[58] := FALSE;
   PLI_WC[59] := FALSE;
   PLI_WC[60] := FALSE;
   PLI_WC[61] := FALSE;
   PLI_WC[62] := FALSE;
   PLI_WC[63] := FALSE;
   PLI_WC[64] := FALSE;
   PLI_WC[65] := FALSE;
   PLI_WC[66] := FALSE;
   PLI_WC[67] := FALSE;
   PLI_WC[68] := FALSE;
   PLI_WC[69] := FALSE;
   PLI_WC[70] := FALSE;
   PLI_WC[71] := FALSE;
   PLI_WC[72] := FALSE;
   PLI_WC[73] := FALSE;
   PLI_WC[74] := FALSE;
   PLI_WC[75] := FALSE;
   PLI_WC[76] := FALSE;
   PLI_WC[77] := FALSE;
   PLI_WC[78] := FALSE;
   PLI_WC[79] := FALSE;
   PLI_WC[80] := FALSE;
   PLI_WC[81] := FALSE;
   PLI_WC[82] := FALSE;
   PLI_WC[83] := FALSE;
   PLI_WC[84] := FALSE;
   PLI_WC[85] := FALSE;
   PLI_WC[86] := FALSE;
   PLI_WC[87] := FALSE;
   PLI_WC[88] := FALSE;
   PLI_WC[89] := FALSE;
   PLI_WC[90] := FALSE;
   PLI_WC[91] := FALSE;
   PLI_WC[92] := FALSE;
   PLI_WC[93] := FALSE;
   PLI_WC[94] := FALSE;
   PLI_WC[95] := FALSE;
   PLI_WC[96] := FALSE;
   PLI_WC[97] := FALSE;
   PLI_WC[98] := FALSE;
   PLI_WC[99] := FALSE;
   PLI_WC[100] := FALSE;
   PLI_WC[101] := FALSE;
   PLI_WC[102] := FALSE;
   PLI_WC[103] := FALSE;
   PLI_WC[104] := FALSE;
   PLI_WC[105] := FALSE;
   PLI_WC[106] := FALSE;
   PLI_WC[107] := FALSE;
   PLI_WC[108] := FALSE;
   PLI_WC[109] := FALSE;
   PLI_WC[110] := FALSE;
   PLI_WC[111] := FALSE;
   PLI_WC[112] := FALSE;
   PLI_WC[113] := FALSE;
   PLI_WC[114] := FALSE;
   PLI_WC[115] := FALSE;
   PLI_WC[116] := FALSE;
   PLI_WC[117] := FALSE;
   PLI_WC[118] := FALSE;
   PLI_WC[119] := FALSE;
   PLI_WC[120] := FALSE;
   PLI_WC[121] := FALSE;
   PLI_WC[122] := FALSE;
   PLI_WC[123] := FALSE;
   PLI_WC[124] := FALSE;
   PLI_WC[125] := FALSE;
   PLI_WC[126] := FALSE;
   PLI_WC[127] := FALSE;
   PLI_WC[128] := FALSE;
   PLI_WC[129] := FALSE;
   PLI_WC[130] := FALSE;
   PLI_WC[131] := FALSE;
   PLI_WC[132] := FALSE;
   PLI_WC[133] := FALSE;
   PLI_WC[134] := FALSE;
   PLI_WC[135] := FALSE;
   PLI_WC[136] := FALSE;
   PLI_WC[137] := FALSE;
   PLI_WC[138] := FALSE;
   PLI_WC[139] := FALSE;
   PLI_WC[140] := FALSE;
   PLI_WC[141] := FALSE;
   PLI_WC[142] := FALSE;
   PLI_WC[143] := FALSE;
   PLI_WC[144] := FALSE;
   PLI_WC[145] := FALSE;
   PLI_WC[146] := FALSE;
   PLI_WC[147] := FALSE;
   PLI_WC[148] := FALSE;
   PLI_WC[149] := FALSE;
   PLI_WC[150] := FALSE;
   PLI_II[1] := FALSE;
   PLI_II[2] := FALSE;
   PLI_II[3] := FALSE;
   PLI_II[4] := FALSE;
   PLI_II[5] := FALSE;
   PLI_II[6] := FALSE;
   PLI_II[7] := FALSE;
   PLI_II[8] := FALSE;
   PLI_II[9] := FALSE;
   PLI_II[10] := FALSE;
   PLI_II[11] := FALSE;
   PLI_II[12] := FALSE;
   PLI_II[13] := FALSE;
   PLI_II[14] := FALSE;
   PLI_II[15] := FALSE;
   PLI_II[16] := FALSE;
   PLI_II[17] := FALSE;
   PLI_II[18] := FALSE;
   PLI_II[19] := FALSE;
   PLI_II[20] := FALSE;
   PLI_II[21] := FALSE;
   PLI_II[22] := FALSE;
   PLI_II[23] := FALSE;
   PLI_II[24] := FALSE;
   PLI_II[25] := FALSE;
   PLI_II[26] := FALSE;
   PLI_II[27] := FALSE;
   PLI_II[28] := FALSE;
   PLI_II[29] := FALSE;
   PLI_II[30] := FALSE;
   PLI_II[31] := FALSE;
   PLI_II[32] := FALSE;
   PLI_II[33] := FALSE;
   PLI_II[34] := FALSE;
   PLI_II[35] := FALSE;
   PLI_II[36] := FALSE;
   PLI_II[37] := FALSE;
   PLI_II[38] := FALSE;
   PLI_II[39] := FALSE;
   PLI_II[40] := FALSE;
   PLI_II[41] := FALSE;
   PLI_II[42] := FALSE;
   PLI_II[43] := FALSE;
   PLI_II[44] := FALSE;
   PLI_II[45] := FALSE;
   PLI_II[46] := FALSE;
   PLI_II[47] := FALSE;
   PLI_II[48] := FALSE;
   PLI_II[49] := FALSE;
   PLI_II[50] := FALSE;
   PLI_II[51] := FALSE;
   PLI_II[52] := FALSE;
   PLI_II[53] := FALSE;
   PLI_II[54] := FALSE;
   PLI_II[55] := FALSE;
   PLI_II[56] := FALSE;
   PLI_II[57] := FALSE;
   PLI_II[58] := FALSE;
   PLI_II[59] := FALSE;
   PLI_II[60] := FALSE;
   PLI_II[61] := FALSE;
   PLI_II[62] := FALSE;
   PLI_II[63] := FALSE;
   PLI_II[64] := FALSE;
   PLI_II[65] := FALSE;
   PLI_II[66] := FALSE;
   PLI_II[67] := FALSE;
   PLI_II[68] := FALSE;
   PLI_II[69] := FALSE;
   PLI_II[70] := FALSE;
   PLI_II[71] := FALSE;
   PLI_II[72] := FALSE;
   PLI_II[73] := FALSE;
   PLI_II[74] := FALSE;
   PLI_II[75] := FALSE;
   PLI_II[76] := FALSE;
   PLI_II[77] := FALSE;
   PLI_II[78] := FALSE;
   PLI_II[79] := FALSE;
   PLI_II[80] := FALSE;
   PLI_II[81] := FALSE;
   PLI_II[82] := FALSE;
   PLI_II[83] := FALSE;
   PLI_II[84] := FALSE;
   PLI_II[85] := FALSE;
   PLI_II[86] := FALSE;
   PLI_II[87] := FALSE;
   PLI_II[88] := FALSE;
   PLI_II[89] := FALSE;
   PLI_II[90] := FALSE;
   PLI_II[91] := FALSE;
   PLI_II[92] := FALSE;
   PLI_II[93] := FALSE;
   PLI_II[94] := FALSE;
   PLI_II[95] := FALSE;
   PLI_II[96] := FALSE;
   PLI_II[97] := FALSE;
   PLI_II[98] := FALSE;
   PLI_II[99] := FALSE;
   PLI_II[100] := FALSE;
   PLI_II[101] := FALSE;
   PLI_II[102] := FALSE;
   PLI_II[103] := FALSE;
   PLI_II[104] := FALSE;
   PLI_II[105] := FALSE;
   PLI_II[106] := FALSE;
   PLI_II[107] := FALSE;
   PLI_II[108] := FALSE;
   PLI_II[109] := FALSE;
   PLI_II[110] := FALSE;
   PLI_II[111] := FALSE;
   PLI_II[112] := FALSE;
   PLI_II[113] := FALSE;
   PLI_II[114] := FALSE;
   PLI_II[115] := FALSE;
   PLI_II[116] := FALSE;
   PLI_II[117] := FALSE;
   PLI_II[118] := FALSE;
   PLI_II[119] := FALSE;
   PLI_II[120] := FALSE;
   PLI_II[121] := FALSE;
   PLI_II[122] := FALSE;
   PLI_II[123] := FALSE;
   PLI_II[124] := FALSE;
   PLI_II[125] := FALSE;
   PLI_II[126] := FALSE;
   PLI_II[127] := FALSE;
   PLI_II[128] := FALSE;
   PLI_II[129] := FALSE;
   PLI_II[130] := FALSE;
   PLI_II[131] := FALSE;
   PLI_II[132] := FALSE;
   PLI_II[133] := FALSE;
   PLI_II[134] := FALSE;
   PLI_II[135] := FALSE;
   PLI_II[136] := FALSE;
   PLI_II[137] := FALSE;
   PLI_II[138] := FALSE;
   PLI_II[139] := FALSE;
   PLI_II[140] := FALSE;
   PLI_II[141] := FALSE;
   PLI_II[142] := FALSE;
   PLI_II[143] := FALSE;
   PLI_II[144] := FALSE;
   PLI_II[145] := FALSE;
   PLI_II[146] := FALSE;
   PLI_II[147] := FALSE;
   PLI_II[148] := FALSE;
   PLI_II[149] := FALSE;
   PLI_II[150] := FALSE;
   PLI_HA[1] := TRUE;
   PLI_HA[2] := TRUE;
   PLI_HA[3] := TRUE;
   PLI_HA[4] := TRUE;
   PLI_HA[5] := TRUE;
   PLI_HA[6] := TRUE;
   PLI_HA[7] := TRUE;
   PLI_HA[8] := TRUE;
   PLI_HA[9] := TRUE;
   PLI_HA[10] := TRUE;
   PLI_HA[11] := TRUE;
   PLI_HA[12] := TRUE;
   PLI_HA[13] := TRUE;
   PLI_HA[14] := TRUE;
   PLI_HA[15] := TRUE;
   PLI_HA[16] := TRUE;
   PLI_HA[17] := TRUE;
   PLI_HA[18] := TRUE;
   PLI_HA[19] := TRUE;
   PLI_HA[20] := TRUE;
   PLI_HA[21] := TRUE;
   PLI_HA[22] := TRUE;
   PLI_HA[23] := TRUE;
   PLI_HA[24] := TRUE;
   PLI_HA[25] := TRUE;
   PLI_HA[26] := TRUE;
   PLI_HA[27] := TRUE;
   PLI_HA[28] := TRUE;
   PLI_HA[29] := TRUE;
   PLI_HA[30] := TRUE;
   PLI_HA[31] := TRUE;
   PLI_HA[32] := TRUE;
   PLI_HA[33] := TRUE;
   PLI_HA[34] := TRUE;
   PLI_HA[35] := TRUE;
   PLI_HA[36] := TRUE;
   PLI_HA[37] := TRUE;
   PLI_HA[38] := TRUE;
   PLI_HA[39] := TRUE;
   PLI_HA[40] := TRUE;
   PLI_HA[41] := TRUE;
   PLI_HA[42] := TRUE;
   PLI_HA[43] := TRUE;
   PLI_HA[44] := TRUE;
   PLI_HA[45] := TRUE;
   PLI_HA[46] := TRUE;
   PLI_HA[47] := TRUE;
   PLI_HA[48] := TRUE;
   PLI_HA[49] := TRUE;
   PLI_HA[50] := TRUE;
   PLI_HA[51] := TRUE;
   PLI_HA[52] := TRUE;
   PLI_HA[53] := TRUE;
   PLI_HA[54] := TRUE;
   PLI_HA[55] := TRUE;
   PLI_HA[56] := TRUE;
   PLI_HA[57] := TRUE;
   PLI_HA[58] := TRUE;
   PLI_HA[59] := TRUE;
   PLI_HA[60] := TRUE;
   PLI_HA[61] := TRUE;
   PLI_HA[62] := TRUE;
   PLI_HA[63] := TRUE;
   PLI_HA[64] := TRUE;
   PLI_HA[65] := TRUE;
   PLI_HA[66] := TRUE;
   PLI_HA[67] := TRUE;
   PLI_HA[68] := TRUE;
   PLI_HA[69] := TRUE;
   PLI_HA[70] := TRUE;
   PLI_HA[71] := TRUE;
   PLI_HA[72] := TRUE;
   PLI_HA[73] := TRUE;
   PLI_HA[74] := TRUE;
   PLI_HA[75] := TRUE;
   PLI_HA[76] := TRUE;
   PLI_HA[77] := TRUE;
   PLI_HA[78] := TRUE;
   PLI_HA[79] := TRUE;
   PLI_HA[80] := TRUE;
   PLI_HA[81] := TRUE;
   PLI_HA[82] := TRUE;
   PLI_HA[83] := TRUE;
   PLI_HA[84] := TRUE;
   PLI_HA[85] := TRUE;
   PLI_HA[86] := TRUE;
   PLI_HA[87] := TRUE;
   PLI_HA[88] := TRUE;
   PLI_HA[89] := TRUE;
   PLI_HA[90] := TRUE;
   PLI_HA[91] := TRUE;
   PLI_HA[92] := TRUE;
   PLI_HA[93] := TRUE;
   PLI_HA[94] := TRUE;
   PLI_HA[95] := TRUE;
   PLI_HA[96] := TRUE;
   PLI_HA[97] := TRUE;
   PLI_HA[98] := TRUE;
   PLI_HA[99] := TRUE;
   PLI_HA[100] := TRUE;
   PLI_HA[101] := TRUE;
   PLI_HA[102] := TRUE;
   PLI_HA[103] := TRUE;
   PLI_HA[104] := TRUE;
   PLI_HA[105] := TRUE;
   PLI_HA[106] := TRUE;
   PLI_HA[107] := TRUE;
   PLI_HA[108] := TRUE;
   PLI_HA[109] := TRUE;
   PLI_HA[110] := TRUE;
   PLI_HA[111] := TRUE;
   PLI_HA[112] := TRUE;
   PLI_HA[113] := TRUE;
   PLI_HA[114] := TRUE;
   PLI_HA[115] := TRUE;
   PLI_HA[116] := TRUE;
   PLI_HA[117] := TRUE;
   PLI_HA[118] := TRUE;
   PLI_HA[119] := TRUE;
   PLI_HA[120] := TRUE;
   PLI_HA[121] := TRUE;
   PLI_HA[122] := TRUE;
   PLI_HA[123] := TRUE;
   PLI_HA[124] := TRUE;
   PLI_HA[125] := TRUE;
   PLI_HA[126] := TRUE;
   PLI_HA[127] := TRUE;
   PLI_HA[128] := TRUE;
   PLI_HA[129] := TRUE;
   PLI_HA[130] := TRUE;
   PLI_HA[131] := TRUE;
   PLI_HA[132] := TRUE;
   PLI_HA[133] := TRUE;
   PLI_HA[134] := TRUE;
   PLI_HA[135] := TRUE;
   PLI_HA[136] := TRUE;
   PLI_HA[137] := TRUE;
   PLI_HA[138] := TRUE;
   PLI_HA[139] := TRUE;
   PLI_HA[140] := TRUE;
   PLI_HA[141] := TRUE;
   PLI_HA[142] := TRUE;
   PLI_HA[143] := TRUE;
   PLI_HA[144] := TRUE;
   PLI_HA[145] := TRUE;
   PLI_HA[146] := TRUE;
   PLI_HA[147] := TRUE;
   PLI_HA[148] := TRUE;
   PLI_HA[149] := TRUE;
   PLI_HA[150] := TRUE;

END_DATA_BLOCK

